// TwinCAT 3 PLC project ukazkaPlc
// Title: ukazkaPlc
// Company: TcOpen.MTS
// ProjectVersion: 0.6.0.913
// ProgramVersion: 3.1.4023.0
// libraries:
//   Tc2_Standard, * (Beckhoff Automation GmbH)
//   Tc2_System, * (Beckhoff Automation GmbH)
//   Tc3_Module, * (Beckhoff Automation GmbH)
//   TcoAbbRobotics, 0.11.0.71 (Vortex.Library)
//   TcoAbstractions, 0.11.0.71 (Vortex.Library)
//   TcoAimTtiPowerSupply, 0.11.0.71 (Vortex.Library)
//   TcoCognexVision, 0.11.0.71 (Vortex.Library)
//   TcoCore, 0.11.0.71 (Vortex.Library)
//   TcoData, 0.11.0.71 (Vortex.Library)
//   TcoDrivesBeckhoff, 0.11.0.71 (Vortex.Library)
//   TcoElements, 0.11.0.71 (Vortex.Library)
//   TcoInspectors, 0.11.0.71 (Vortex.Library)
//   TcoIo, 0.11.0.71 (Vortex.Library)
//   TcoKukaRobotics, 0.11.0.71 (Vortex.Library)
//   TcoMitsubishiRobotics, 0.11.0.71 (Vortex.Library)
//   TcoPneumatics, 0.11.0.71 (Vortex.Library)
//   TcoRexrothPress, 0.11.0.71 (Vortex.Library)
//   TcoTixonFeeding, 0.11.0.71 (Vortex.Library)
//   TcoUrRobotics, 0.11.0.71 (Vortex.Library)
//   TcoUtilities, 0.11.0.71 (Vortex.Library)
// project tree:
//   Abstractions/Components/ArrayRenderingExample/ SampleArrayToRender.TcDUT, SampleDataItem.TcDUT
//   Abstractions/Components/MtsFeeding/ TcoFeedingSequenceTask.TcPOU, TcoPlsPaletizator.TcPOU, TcoPlsPaletizator_Components.TcDUT, TcoPlsPaletizator_Config_v_1_x_x.TcDUT, TcoPlsPaletizator_Control_v_1_x_x.TcDUT, TcoPlsPaletizator_Status_v_1_x_x.TcDUT
//   Abstractions/Components/WrappedComponent/ WrappedComponentExample.TcPOU, WrappedComponentExample_Config.TcDUT, WrappedComponentExample_Control.TcDUT, WrappedComponentExample_Status.TcDUT, WrappedComponentsExample.TcDUT
//   Abstractions/CUBase/ CuBaseRecurringFail.TcDUT, CuBaseRecurringFailures.TcDUT, CUBase.TcPOU, CUBaseStatusInfo.TcDUT, CUBaseSettings.TcDUT, CUComponentsBase.TcDUT, ICUBase.TcIO, ICUTask.TcIO, OperatorInfo.TcDUT
//   Abstractions/CUBase/Data/ CuHeader.TcDUT, CUProcessDataBase.TcDUT, CUTechnologicalDataBase.TcDUT, eCUMode.TcDUT, eCUState.TcDUT, eDataEntityInvokeType.TcDUT, EntityHeader.TcDUT
//   Abstractions/CUBase/RemoteTasks/ ProductionPlaner.TcPOU
//   Abstractions/CUBase/Tasks/ CUBaseAutomat.TcPOU, CUBaseSuspend.TcPOU, CUBaseGround.TcPOU, CUBaseRecover.TcPOU
//   Abstractions/Generic/NotificationPanel/ NotificationPanel.TcPOU, NotificationPanelInfo.TcDUT
//   Abstractions/Safety/ControlButtons/ TcoControlButtons.TcPOU, ITcoControlButtons.TcIO, TcoControledZone_Info.TcDUT
//   Abstractions/Safety/ControlledZone/ TcoControlledZoneActionTask.TcPOU, TcoControlledZone.TcPOU, TcoControlledZone_Config.TcDUT, TcoControlledZone_Status.TcDUT
//   Abstractions/Safety/ControlVoltage/ ITcoControlVoltage.TcIO, TcoControlVoltage.TcPOU
//   Abstractions/Safety/DoorCircuit/ TcoDoorCircuit_Status.TcDUT, TcoDoorCircuit_Config.TcDUT, TcoDoorCircuit.TcPOU, ITcoDoorCircuit.TcIO
//   Abstractions/Safety/Doors/ ITcoDoorLock.TcIO, TcoStandardDoor.TcPOU, TcoBasicDoor.TcPOU
//   Abstractions/Safety/Estop/ TcoEmergencyStop.TcPOU
//   Abstractions/Safety/KeyMode/ TcoKeyMode_Config.TcDUT, TcoKeyMode_Status.TcDUT, TcoKeyMode.TcPOU, ITcoKeyMode.TcIO
//   Abstractions/Safety/KeyNormalService/ TcoKeyNormalService.TcPOU, ITcoKeyNormalSevice.TcIO
//   Abstractions/TcoCore/ CycleTimeAnalitics.TcDUT, TcoInnerTask.TcPOU, TcoTaskedSequencer.TcPOU, TcoTaskedService.TcPOU
//   Abstractions/Technology/ eStations.TcDUT
//   / MAIN.TcPOU, PlcTask.TcTTO
//   Technology/CU00x/Automat/ CU00xAutomatParalell_1_Task.TcPOU, CU00xAutomatTask.TcPOU
//   Technology/CU00x/Components/ CU00xExamplesOfComponents.TcDUT, CU00xComponents.TcDUT
//   Technology/CU00x/Data/ CU00xTechnologicalData.TcDUT, CU00xDialogContent.TcPOU, CU00xProcessData.TcDUT
//   Technology/CU00x/Ground/ CU00xGroundTask.TcPOU
//   Technology/CU00x/Manual/ CU00xManualTask.TcPOU
//   Technology/CU00x/Positions/ CU00xTestMultiPositions.TcPOU, Cu00xTestPositions.TcPOU
//   Technology/CU00x/Safety/Suspend/ CU00xSuspendTask.TcPOU
//   Technology/CU00x/Safety/Recover/ CU00xRecoverTask.TcPOU
//   Technology/Data/ ProcessData.TcDUT, ProcessDataManager.TcPOU, TcoEntityBase.TcDUT, TechnologicalDataManager.TcPOU, TechnologyData.TcDUT
//   Technology/CU00x/ CU00x.TcPOU
//   Technology/ Technology.TcPOU, TechnologyComponents.TcDUT (not stored)
//   DUTs/IO/PDOs/ Device_State_F0482DC3.TcDUT, Device_Control_6258066A.TcDUT, Inputs_23559BB0.TcDUT, Outputs_FC2FACAD.TcDUT, Modules_85784B27.TcDUT, Channel_830843C1.TcDUT, Channel_42CA91F7.TcDUT
//   DUTs/IO/Boxes/ EK1200_013D0B49.TcDUT, EK1122_1FC0878B.TcDUT, AES_510494FB.TcDUT, EPP1322_1FC0878B.TcDUT, EPP1809_32157CFD.TcDUT, EPP1008_78E8D3DD.TcDUT, EL1809_32157CFD.TcDUT, EL2809_2B6483BD.TcDUT, EL9011_D65D3D32.TcDUT
//   DUTs/IO/Devices/ SyncUnitTasks_4BE01469.TcDUT, SyncUnits_67D36DDA.TcDUT
//   DUTs/IO/Topology/ EK_E812B8FA.TcDUT, EC_4E5C738F.TcDUT, EC_245FBB9A.TcDUT
//   GVLs/ GVL_iXlinker.TcGVL
// real-time tasks:
//   TASK PlcTask: cycle T#10ms, priority 20, ADS port 350
//   TASK PlcTask1: cycle T#10ms, priority 21, ADS port 351
// I/O:
//   DEVICE EC1 (disabled), AmsNetId 172.20.21.220.7.1
//     (EK1200) [EK1200-5000 EtherCAT Power supply (2A E-Bus)]
//       EC (EK1122) [EK1122 2 port EtherCAT junction]
//       PN (EL6631) [EL6631 PROFINET IO Controller]
//       IA1 (EL1809) [EL1809 16Ch. Dig. Input 24V, 3ms]
//       QA1 (EL2809) [EL2809 16Ch. Dig. Output 24V, 0.5A]
//       Term 6 (EL4004) [EL4004 4Ch. Ana. Output 0-10V, 12bit]
//       Term 7 (EL7342) [EL7342 2Ch. DC motor output stage (50V, 3.5A)]
//       Term 8 (EL4004) [EL4004 4Ch. Ana. Output 0-10V, 12bit]
//       Term 9 (EL6001) [EL6001 Interface (RS232)]
//       Term 13 (EL9011) [EL9011 End Terminal]
//   DEVICE EC (disabled), AmsNetId 172.20.21.220.2.1
//     EC [EK1200-5000 EtherCAT Power supply (2A E-Bus)]
//       EK [EK1122 2 port EtherCAT junction]
//         PNEU [AES Fieldbus Coupler Gen2]
//           modules: Modules
//         AB [EPP1322-0001 3 port EtherCAT P gateway]
//         AB21 [EPP1809-0021 16 Ch. Dig. Input 24V, 3ms, M8]
//         AB22 [EPP1809-0021 16 Ch. Dig. Input 24V, 3ms, M8]
//         AB23 [EPP1008-0001 8 Ch. Dig. Input 24V, 3ms, M8]
//         AB24 [EPP1008-0001 8 Ch. Dig. Input 24V, 3ms, M8]
//       IA1 [EL1809 16Ch. Dig. Input 24V, 3ms]
//       QA1 [EL2809-0015 16Ch. Dig. Output 24V DC, 0.35A, not short-circuit proof]
//       Term 11 (EL9011) [EL9011 End Terminal]

CONFIGURATION ukazkaPlc
    RESOURCE PLC ON TwinCAT3
        TASK PlcTask(INTERVAL := T#10ms, PRIORITY := 20);
        PROGRAM MAIN WITH PlcTask : MAIN;
    END_RESOURCE
END_CONFIGURATION

// ---- Abstractions/Components/ArrayRenderingExample/SampleArrayToRender.TcDUT
TYPE SampleArrayToRender :
STRUCT
	Data	:	ARRAY  [0..100] OF SampleDataItem;
END_STRUCT
END_TYPE

// ---- Abstractions/Components/ArrayRenderingExample/SampleDataItem.TcDUT
TYPE SampleDataItem :
STRUCT
 	Measured : BOOL;
    Overrided : BOOL;
    Marginal : BOOL;
    FinalResults : BOOL;
END_STRUCT
END_TYPE

// ---- Abstractions/Components/MtsFeeding/TcoPlsPaletizator_Components.TcDUT
TYPE TcoPlsPaletizator_Components EXTENDS TcoCore.TcoStruct:
STRUCT
	
	{attribute wpf [Container(Layout.Stack)]}
	{attribute addProperty Name "(I1) <#Pritomnost blistra v presuvaci#>"}
	I1_PresentBlisterEntry : TcoElements.TcoDi(THISSTRUCT);
	
	{attribute addProperty Name "(I2) <#Pritomnost medzery medzi blistrami#>"}
	I2_PresentBlisterEntryEmptySpace : TcoElements.TcoDi(THISSTRUCT);
	
	{attribute addProperty Name "(I3) <#Zasobik blistrov prazdny#>"}
	I3_PresentBlistersInBufferEmpty : TcoElements.TcoDi(THISSTRUCT);

	
	{attribute addProperty Name "(I4) <#Pritomnost blistra v pracovnej pozicii#>"}
	I4_PresentBlisterInWorkingPos : TcoElements.TcoDi(THISSTRUCT);
		
	{attribute addProperty Name "(I5) <#Vystupny blister neje v sklzovom dopravniku#>"}
	I5_OutBlistersIsThrowedCorrectly : TcoElements.TcoDi(THISSTRUCT);
	
	{attribute addProperty Name "(I6) <#Vystupny blister snimanie vo vytahu#>"}
	I6_OutBlistersLisftSignal : TcoElements.TcoDi(THISSTRUCT);
	
	{attribute addProperty Name "(I7) <#Vystupny blister je nad Bufferom#>"}
	I7_OutBlistersIsAboveOutBuffer : TcoElements.TcoDi(THISSTRUCT);
	
	{attribute addProperty Name "(I8) <#Vystupny zasobnik je plny#>"}
	I8_OutBlistersBufferIsFull : TcoElements.TcoDi(THISSTRUCT);
	
	
	{attribute wpf [Container(Layout.Stack)]}
	{attribute addProperty Name "(P1) <#Vertikalny prisun vstupnych blistrov#>"}
	P1_VerticalSepareEntryBlisters : TcoPneumatics.TcoCylinder(THISSTRUCT);
	
	{attribute addProperty Name "(P2) <#Vertikalny prisun vstupnych blistrov#>"}
	P2_VerticalSepareEntryBlisters : TcoPneumatics.TcoCylinder(THISSTRUCT);
	
	{attribute addProperty Name "(P3) (P3.1) <#Horizontalny prisun vstupnych blistrov#>"}
	P3_HorizontalSepareEntryBlisters : TcoPneumatics.TcoDoubleCylinder(THISSTRUCT);
		
	{attribute addProperty Name "(P4) <#Prisun vstupneho blistra#>"}
	P4_FeedEntryBlister :TcoPneumatics.TcoCylinder(THISSTRUCT);
	
	{attribute addProperty Name "(P5) (P5.1)<#Horizontalny prisun vystupnych blistrov#>"}
	P5_HorizontalSepareOutBlisters : TcoPneumatics.TcoDoubleCylinder(THISSTRUCT);
	
	{attribute addProperty Name "(P6)<#Vertikalny prisun vystupnych blistrov#>"}
	P6_VerticalSepareOutBlister : TcoPneumatics.TcoCylinder(THISSTRUCT);
	
	{attribute addProperty Name "(P7) <#Podopretie vstupneho blistra#>"}
	P7_SupportEntryBlister : TcoPneumatics.TcoCylinder(THISSTRUCT);
	
	{attribute addProperty Name "(P8) (P8.1) <#Upevnenie zboku vstupneho blistra#>"}
	P8_FixEntryBlisterSide : TcoPneumatics.TcoDoubleCylinder(THISSTRUCT);
	
	{attribute addProperty Name "(P9) (P9.1) <#Zamknutue zhora vstupneho blistra#>"}
	P9_LockEntryBlisterTop : TcoPneumatics.TcoDoubleCylinder(THISSTRUCT);
	
	{attribute addProperty Name "(P10) (P10.1)<#Odelovac blistrov na vstupe#>"}
	P10_HoldEntrySepareOutBlister : TcoPneumatics.TcoDoubleCylinder(THISSTRUCT);
	
	
	
	{attribute wpf [Container(Layout.Stack,"Vseobecne")]}
	
	{attribute addProperty Name "(Q1) <#Signalizacia upozornenia R#>"}
	Q1_AttentionSignalisationR : TcoElements.TcoDo(THISSTRUCT);
	{attribute addProperty Name "(Q2) <#Signalizacia upozornenia G#>"}
	Q2_AttentionSignalisationG : TcoElements.TcoDo(THISSTRUCT);
	{attribute addProperty Name "(Q3) <#Signalizacia upozornenia B#>"}
	Q3_AttentionSignalisationB : TcoElements.TcoDo(THISSTRUCT);

	
	
END_STRUCT
END_TYPE

// ---- Abstractions/Components/MtsFeeding/TcoPlsPaletizator_Config_v_1_x_x.TcDUT
TYPE
    TcoPlsPaletizator_Config_v_1_x_x EXTENDS TcoCore.TcoStruct :
    STRUCT

	
        {attribute addProperty Name "<#Stabilizacny cas#>"}
		StabilisationTime : TIME :=T#500MS;
		{attribute addProperty Name "<#Blink period#>"}
		BlinkTime : TIME := T#500MS;
		
        {attribute addProperty Name "<#Zamykanie blistra zhora neaktive (P9)(P9.1)je nepritomne#>"}
		LockBlisterInPickPosInactive : BOOL;
		
		{attribute addProperty Name "<#Oddelovanie blistrov na vstupe neaktive (P10)(P10.1)je nepritomne#>"}
		SepareBlistersAtEntryInactive : BOOL;
    END_STRUCT
END_TYPE

// ---- Abstractions/Components/MtsFeeding/TcoPlsPaletizator_Control_v_1_x_x.TcDUT
TYPE TcoPlsPaletizator_Control_v_1_x_x EXTENDS TcoCore.TcoStruct:
STRUCT

		
END_STRUCT
END_TYPE

// ---- Abstractions/Components/MtsFeeding/TcoPlsPaletizator_Status_v_1_x_x.TcDUT
TYPE
    TcoPlsPaletizator_Status_v_1_x_x EXTENDS TcoCore.TcoStruct :
    STRUCT

        ActionDescription : STRING;
        SafeCondition : BOOL;
		EntryBufferEmpty:BOOL;
        BlisterReady : BOOL;
        OutBufferFull : BOOL;
    END_STRUCT
END_TYPE

// ---- Abstractions/Components/WrappedComponent/WrappedComponentExample_Config.TcDUT
TYPE
    WrappedComponentExample_Config EXTENDS TcoCore.TcoStruct :
    STRUCT

        VacuumReachedStabilisation : TIME := T#100MS;
        VacuumPushTime : TIME := T#100MS;
    END_STRUCT
END_TYPE

// ---- Abstractions/Components/WrappedComponent/WrappedComponentExample_Control.TcDUT
TYPE WrappedComponentExample_Control EXTENDS TcoCore.TcoStruct:
STRUCT

		Setpoint:INT;
		
END_STRUCT
END_TYPE

// ---- Abstractions/Components/WrappedComponent/WrappedComponentExample_Status.TcDUT
TYPE WrappedComponentExample_Status EXTENDS TcoCore.TcoStruct:
STRUCT

		ProgressThrow:INT;
		ActionDescription:STRING;
END_STRUCT
END_TYPE

// ---- Abstractions/Components/WrappedComponent/WrappedComponentsExample.TcDUT
TYPE WrappedComponentsExample EXTENDS TcoCore.TcoStruct:
STRUCT
	
		{attribute addProperty Name "Vacuum Reached"}
		VacuumReached : TcoElements.TcoDi(THISSTRUCT);
		{attribute addProperty Name "Vacuum On"}
		VacuumOn : TcoElements.TcoDo(THISSTRUCT);
		{attribute addProperty Name "Vacuum Push"}
		VacuumPush : TcoElements.TcoDo(THISSTRUCT);
		
		{attribute addProperty Name "Gripper"}
		Gripper : TcoPneumatics.TcoCylinder(THISSTRUCT);
  
		{attribute addProperty Name "Manipulator"}
		Manipulator : TcoDrivesBeckhoff.TcoMultiAxis(THISSTRUCT);

		{attribute addProperty Name "Component Picked"}
		PresenceInGripper : TcoElements.TcoDi(THISSTRUCT);

	
	
END_STRUCT
END_TYPE

// ---- Abstractions/CUBase/CuBaseRecurringFail.TcDUT
TYPE CuBaseRecurringFail :
STRUCT
	Reached:BOOL;
	Result:TcoComprehensiveResult;
	Counter:UINT;
	
	
	
	
	
END_STRUCT
END_TYPE

// ---- Abstractions/CUBase/CuBaseRecurringFailures.TcDUT
TYPE CuBaseRecurringFailures EXTENDS TcoCore.TcoStruct : 
	STRUCT
   		AnyRecurringFails : CuBaseRecurringFail;
    	SameRecurringFails : CuBaseRecurringFail;
	END_STRUCT
END_TYPE

// ---- Abstractions/CUBase/CUBaseStatusInfo.TcDUT
TYPE
    CUBaseStatusInfo EXTENDS TcoCore.TcoStruct :
    STRUCT
     Mode                   : eCUMode;
     CurrentTaskDescription : STRING;
     CurrentUid             : INT;
     CurrentOperation       : STRING(255);
     CurrentCycleTime       : TIME;
	 AverageCycleTime       : TIME;
     CurrentIsInStepMode    : BOOL;
     CurrentCleanCycleTime  : TIME;
	 AverageCleanCycleTime  : TIME;
     State	                : eCUState;
     InSavingEnergy         : BOOL;
    END_STRUCT
END_TYPE

// ---- Abstractions/CUBase/CUBaseSettings.TcDUT
TYPE CUBaseSettings EXTENDS TcoCore.TcoStruct : STRUCT
    DeafultCycleTime : TIME;
    WarningCycleTime : TIME;
    ErrorCycleTime : TIME;
    SaveEnergyTime : TIME;
    AnyRecurringFailure : UINT;
    SameRecurringFailure : UINT;
END_STRUCT
END_TYPE

// ---- Abstractions/CUBase/CUComponentsBase.TcDUT
TYPE
    CUComponentsBase EXTENDS TcoCore.TcoStruct :
    STRUCT
       
    END_STRUCT
END_TYPE

// ---- Abstractions/CUBase/Data/CuHeader.TcDUT
TYPE CuHeader EXTENDS TcoCore.TcoStruct :
STRUCT
	{attribute addProperty Name "<#Next on Passed#>"}
	NextOnPassed : eStations;
	{attribute addProperty Name "<#Next on Failed#>"}
	NextOnFailed : eStations;
	{attribute clr [RenderIgnore("Control", "ShadowControl")]}
	{attribute addProperty Name "<#Cycle time#>"}
	CycleTime : TIME;
	{attribute clr [RenderIgnore("Control", "ShadowControl")]}
	{attribute addProperty Name "<#Clean loop time#>"}
	CleanLoopTime : TIME;
	{attribute clr [RenderIgnore("Control", "ShadowControl")]}
	{attribute addProperty Name "<#Operation started#>"}
	OperationsStarted : DT;
	{attribute clr [RenderIgnore("Control", "ShadowControl")]}
	{attribute addProperty Name "<#Operation ended#>"}
	OperationsEnded : DT;	
	{attribute clr [RenderIgnore("Control", "ShadowControl")]}
	{attribute addProperty Name "<#Operator#>"}
	Operator :STRING;	
END_STRUCT
END_TYPE

// ---- Abstractions/CUBase/Data/CUProcessDataBase.TcDUT
{attribute clr [Container(Layout.Stack)]}
{attribute clr [Group(Layout.Scroll)]}
TYPE CUProcessDataBase EXTENDS TcoCore.TcoStruct :
STRUCT
	{attribute wpf [Container(Layout.Stack)]}
	{attribute wpf [Group(Layout.GroupBox)]}
	Header : CuHeader := (Parent := THISSTRUCT);
END_STRUCT
END_TYPE

// ---- Abstractions/CUBase/Data/CUTechnologicalDataBase.TcDUT
{attribute clr [Container(Layout.Stack)]}
{attribute clr [Group(Layout.Scroll)]}
TYPE CUTechnologicalDataBase EXTENDS TcoCore.TcoStruct :
STRUCT
	{attribute wpf [Container(Layout.Stack,"General")]}
	{attribute wpf [Group(Layout.GroupBox)]}
	{attribute addProperty Name "<#Cycle time#> - <#Nominal#>"}
	IdealCycleTime   : TIME;
	
	
	{attribute addProperty Name "<#Cycle time#> - <#Warning#>"}
	WarningCycleTime : TIME;
    
	{attribute addProperty Name "<#Cycle time#> - <#Error#>"}
	ErrorCycleTime   : TIME;

	
	{attribute addProperty Name "<#Step time#> - <#Warning#>"}
	WarningStepAlarmTime : TIME;
    
	{attribute addProperty Name "<#Step time#> - <#Error#>"}
	ErrorStepAlarmTime   : TIME;
	
	{attribute addProperty Name "<#Energy saving mode - Inactivity time#>"}
	TimeToEntryEnergySavingMode : TIME;
	
	
	
	(*~
	<docu>
		<summary>
			The maximum allowed number of the any (arbitrary) recuring (consecutive)  failures.
		</summary>			
	</docu>	
	~*)
	{attribute addProperty Name "<#Max allowed number of any recurring failures (consecutive)#>"}
	AnyRecurringFailure   : UINT;
	
	

	(*~
	<docu>
		<summary>
			The maximum allowed number of the same (identical) recuring (consecutive) failures. 
		</summary>			
	</docu>	
	~*)
	{attribute addProperty Name "<#Max allowed number of same recurring failures (consecutive)#>"}
	SameRecurringFailure   : UINT;
	
	
END_STRUCT
END_TYPE

// ---- Abstractions/CUBase/Data/eCUMode.TcDUT
{attribute 'qualified_only'}
{attribute 'strict'}
TYPE
    eCUMode :
    (
        NoMode         := 0,
        GroundMode     := 10,
        GroundModeDone := 15,
        AutomatMode    := 20,
        ManualMode     := 30
    );
END_TYPE

// ---- Abstractions/CUBase/Data/eCUState.TcDUT
{attribute 'qualified_only'}
{attribute 'strict'}
TYPE
    eCUState :
    (
        None       := 0,
        HasWarning := 10,
        HasError   := 20
    );
END_TYPE

// ---- Abstractions/CUBase/Data/eDataEntityInvokeType.TcDUT
{attribute 'qualified_only'}
{attribute 'strict'}
TYPE eDataEntityInvokeType : (
    InvokeAndWaitDone := 0,
    InvokeOnly	 := 10
);
END_TYPE

// ---- Abstractions/CUBase/Data/EntityHeader.TcDUT
{attribute wpf [Container(Layout.Stack)]}
{attribute wpf [Group(Layout.Scroll)]}
{attribute addProperty Name "<#Entity header#>"}
TYPE
    EntityHeader EXTENDS TcoCore.TcoStruct :
    STRUCT
        {attribute addProperty Name "<#Recipe#>"}
        {attribute clr [RenderIgnore("Control", "ShadowControl")]}
        Recipe : STRING(255);
        {attribute addProperty Name "<#Recipe created#>"}
        {attribute clr [RenderIgnore("Control", "ShadowControl")]}
        RecipeCreated : DT;
        {attribute addProperty Name "<#Recipe modified#>"}
        {attribute clr [RenderIgnore("Control", "ShadowControl")]}
        RecipeLastModified : DT;
        {attribute addProperty Name "<#Carrier#>"}
        {attribute clr [RenderIgnore("Control", "ShadowControl")]}
        Carrier : STRING;
        {attribute addProperty Name "<#Reset#>"}
        {attribute clr [RenderIgnore("Control", "ShadowControl")]}
        WasReset : BOOL;
        {attribute addProperty Name "<#Master#>"}
        {attribute clr [RenderIgnore("Control", "ShadowControl")]}
        IsMaster : BOOL;
        {attribute addProperty Name "<#Empty#>"}
        {attribute clr [RenderIgnore("Control", "ShadowControl")]}
        IsEmpty : BOOL;
        {attribute addProperty Name "<#Last station#>"}
        LastStation : eStations;
        {attribute addProperty Name "<#Next station#>"}
        NextStation : eStations;
        {attribute addProperty Name "<#Operations opened#>"}
        OpenOn : eStations;
        {attribute addProperty Name "<#Results#>"}
        Results : TcoInspectors.TcoComprehensiveResult;

        {attribute addProperty Name "<#Reworked#>"}
        {attribute clr [RenderIgnore("Control", "ShadowControl")]}
         WasReworked : BOOL;

        {attribute addProperty Name "<#Last Rework Name#>"}
        {attribute clr [RenderIgnore("Control", "ShadowControl")]}
         LastReworkName : STRING;

        {attribute addProperty Name "<#Rework Count#>"}
        {attribute clr [RenderIgnore("Control", "ShadowControl")]}
        ReworkCount : SINT;

    END_STRUCT
END_TYPE

// ---- Abstractions/CUBase/OperatorInfo.TcDUT
TYPE OperatorInfo EXTENDS TcoCore.TcoStruct :
STRUCT
	UserName : STRING(255);
END_STRUCT
END_TYPE

// ---- Abstractions/Generic/NotificationPanel/NotificationPanelInfo.TcDUT
TYPE NotificationPanelInfo :
STRUCT
	{attribute addProperty Name "<#Control voltage#>"}
	ControlVoltage : BOOL;
	{attribute addProperty Name "<#Air pressure#>"}
	AirPressure : BOOL;
	{attribute addProperty Name "<#Autmatic mode allowed#>"}
	AutomatAllowed : BOOL;
	{attribute addProperty Name "<#Emergency stop#>"}
  	EmergencyStop : BOOL; 
	{attribute addProperty Name "<#Safety doors OK#>"}
  	SafetyDoorOk : BOOL;    
	{attribute addProperty Name "<#Doors closed#>"}
  	DoorClosed : BOOL;  
	{attribute addProperty Name "<#Doors locked#>"}
	DoorLocked : BOOL;
	{attribute addProperty Name "<#Light curtain#>"}
  	LightCurtain : BOOL;
	{attribute addProperty Name "<#Process data#>"}
  	ProcessDataOk : BOOL;
	{attribute addProperty Name "<#Technology data#>"}
  	TechnologyDataOk : BOOL;
END_STRUCT
END_TYPE

// ---- Abstractions/Safety/ControlButtons/TcoControledZone_Info.TcDUT
TYPE TcoControledZone_Info :
STRUCT
	{attribute addProperty Name "<#All#> - <#In automatic#>"}
	AllInAuto            : BOOL;
	
	{attribute addProperty Name "<#All#> - <#Is grounding#>"}
	AllInGrounding       : BOOL;
	
	{attribute addProperty Name "<#All#> - <#In manual#>"}
	AllInManual          : BOOL;
	
	{attribute addProperty Name "<#All#> - <#Idle#>"}
	AllIdle          : BOOL;

	{attribute addProperty Name "<#All#> - <#Grounded#>"}
	AllGrounded          : BOOL;
	
	{attribute addProperty Name "<#All#> - <#In step mode#>"}
	AllInStepMode        : BOOL;
	
	{attribute addProperty Name "<#All#> - <#Recovered#>"}
	AllRecovered        : BOOL;
	
	{attribute addProperty Name "<#All#> - <#Suspended#>"}
	AllSuspended        : BOOL;
	
	{attribute addProperty Name "<#All#> - <#Holding process#>"}
	AllHolding           : BOOL;
	
	{attribute addProperty Name "<#All#> - <#In Inactive or Manual or Grounded#>"}
	AllInactiveOrManualOrGrounded  : BOOL;
	
	{attribute addProperty Name "<#Group#> - <#Any station in automatic mode#>"}
	AnyInAuto            : BOOL;
	
	{attribute addProperty Name "<#Group#> - <#Any station in manual mode#>"}
	AnyInManual          : BOOL;
	
	{attribute addProperty Name "<#Group#> - <#Any station in step mode#>"}
	AnyInStepMode        : BOOL;
	
	{attribute addProperty Name "<#Group#> - <#Any station is grounding#>"}
	AnyGrounding         : BOOL;
	
	{attribute addProperty Name "<#Group#> - <#Any station is holded#>"}
	AnyInHolding         : BOOL;
	
	{attribute addProperty Name "<#Control panel#> - <#All keys in automatic#>"}
	AllKeysAuto          : BOOL;
	
	{attribute addProperty Name "<#Control panel#> - <#All keys in normal#>"}
	AllKeysNormal        : BOOL;
	
	{attribute addProperty Name "<#Control panel#> - <#Any key in manual#>"}
	AnyKeyManual         : BOOL;
	
	{attribute addProperty Name "<#Control panel#> - <#Any key in step#>"}
	AnyKeyStep           : BOOL;
	
	{attribute addProperty Name "<#Control panel#> - <#Any key in service#>"}
	AnyKeyService        : BOOL;
	
	{attribute addProperty Name "<#Control panel#> - <#Any button#> - <#Recover#>"}
	AnyButtonRecover       : BOOL;
	
	{attribute addProperty Name "<#Control panel#> - <#Any button#> - <#Suspend#>"}
	AnyButtonSuspend        : BOOL;
	
	{attribute addProperty Name "<#Control panel#> - <#Any button#> - <#Ground#>"}
	AnyButtonGround      : BOOL;
	
	{attribute addProperty Name "<#Control panel#> - <#Any button#> - <#Auto#>"}
	AnyButtonAuto     : BOOL;
	
	{attribute addProperty Name "<#Deadman#> - <#Any present#>"}
	AnyDeadmanPresent    : BOOL;

END_STRUCT
END_TYPE

// ---- Abstractions/Safety/ControlledZone/TcoControlledZone_Config.TcDUT
TYPE
    TcoControlledZone_Config :
    STRUCT
        MaxControledUnits : USINT := 12;
        MaxControlButtons : USINT := 4;
        MaxKeyMode : USINT := 4;
        MaxKeyNormalService : USINT := 4;
        DoorsLocked : TIME := T#1S;
		AirPressureErrorTime : TIME :=T#5S;
    END_STRUCT
END_TYPE

// ---- Abstractions/Safety/ControlledZone/TcoControlledZone_Status.TcDUT
TYPE TcoControlledZone_Status :
STRUCT
	ActionDescription : STRING(100);	
	State : TcoControledZone_Info;	
	
END_STRUCT
END_TYPE

// ---- Abstractions/Safety/DoorCircuit/TcoDoorCircuit_Status.TcDUT
TYPE TcoDoorCircuit_Status :
STRUCT
	ActionDescription : STRING(100);	
END_STRUCT
END_TYPE

// ---- Abstractions/Safety/DoorCircuit/TcoDoorCircuit_Config.TcDUT
TYPE
    TcoDoorCircuit_Config :
    STRUCT
        InfoTime : TIME := T#2S;
        ErrorTime : TIME := T#0S;
		MaxDoors : USINT:=12;
		MaxLocalDoorsVoltage : USINT:=4;
		MaxLocalVoltage: USINT:=4;
		MaxGlobalVoltage: USINT:=4;
	
    END_STRUCT
END_TYPE

// ---- Abstractions/Safety/KeyMode/TcoKeyMode_Config.TcDUT
TYPE
    TcoKeyMode_Config :
    STRUCT
        SwitKeyStanilisiation : TIME := T#500mS;

	
    END_STRUCT
END_TYPE

// ---- Abstractions/Safety/KeyMode/TcoKeyMode_Status.TcDUT
TYPE TcoKeyMode_Status :
STRUCT
	ActionDescription : STRING(100);	

END_STRUCT
END_TYPE

// ---- Abstractions/TcoCore/CycleTimeAnalitics.TcDUT
TYPE CycleTimeAnalitics :
STRUCT

	{attribute addProperty Name "<#Average cycle time#>"}
	Average:TIME;
	
	{attribute addProperty Name "<#Average clean cycle time#>"}
	AverageCleanCycle:TIME;
	
	{attribute addProperty Name "<#Average cycle time filter constant#>"}
	FilterConstant:UINT:=10;	
	

	
END_STRUCT
END_TYPE

// ---- Abstractions/Technology/eStations.TcDUT
{attribute 'qualified_only'}
{attribute 'strict'}
TYPE
    eStations :
    (
		CU00x := 100,
        ST_1  := 1,
        ST_2  := 2,
        ST_3  := 3,
        ST_4  := 4,
        ST_5  := 5,
        ST_6  := 6,
        ST_7  := 7,
        ST_8  := 8,
        ST_9  := 9,
        ST_10 := 10,
        ST_11 := 11,
        ST_12 := 12,
        ST_13 := 13,
        ST_14 := 14,
        ST_15 := 15,
        ST_16 := 16,
        ST_17 := 17,
        ST_18 := 18,
        ST_19 := 19,
        ST_20 := 20,
        NONE  := 32767
    );
END_TYPE

// ---- Technology/CU00x/Components/CU00xExamplesOfComponents.TcDUT
{attribute wpf [Container(Layout.Stack)]}	
{attribute wpf [Group(Layout.Scroll)]}
TYPE CU00xExamplesOfComponents EXTENDS TcoCore.TcoStruct:
STRUCT
		{attribute wpf [Container(Layout.Stack,"PNEU")]}	
		{attribute addProperty Name "(A1)HORIZONTAL AXIS"}
      	horizontalCylinder : TcoPneumatics.TcoCylinder(THISSTRUCT); 
		{attribute addProperty Name "(A2)VERTICAL AXIS"}
      	verticalCylinder : TcoPneumatics.TcoCylinder(THISSTRUCT); 
		
		{attribute addProperty Name "(A3)DOUBLE "}
      	doubleCylinder : TcoPneumatics.TcoDoubleCylinder(THISSTRUCT); 
		
		{attribute wpf [Container(Layout.Stack,"INPUTS")]}	
		{attribute addProperty Name "PRESENCE ON INSPECTION"}
     	PresenceOnInspection : TcoElements.TcoDi(THISSTRUCT);
		
		{attribute addProperty Name "PRESENCE AT ENTRY CONVEYOR"}
     	PresenceComponentAtEntr: TcoElements.TcoDi(THISSTRUCT);
		
		{attribute addProperty Name "COLISION SENSOR"}
     	ColisonSensorComponent: TcoElements.TcoDi(THISSTRUCT);

		{attribute addProperty Name "CONVEYOR AT ENTRY IS EMPTY"}
     	ConvAtEntryIsEmpty : TcoElements.TcoDi(THISSTRUCT);
		
		{attribute addProperty Name "INSPECTION NOK"}
     	InspectionIsNok : TcoElements.TcoDi(THISSTRUCT);
		

		{attribute wpf [Container(Layout.Stack,"OUTPUTS")]}		
		{attribute addProperty Name "LIGHT ON"}
     	LightOn : TcoElements.TcoDi(THISSTRUCT); 
		
		{attribute addProperty Name "LIGHT OFF"}
     	LightOff : TcoElements.TcoDi(THISSTRUCT);
		{attribute wpf [Container(Layout.Stack,"ANALOGS")]}	
		{attribute addProperty Name "VERIFY SETPOINT"}
     	VerifySetpoint : TcoElements.TcoAi(THISSTRUCT);
		{attribute addProperty Name "SETPOINT"}
     	Setpoint : TcoElements.TcoAo(THISSTRUCT);   
		
		{attribute addProperty Name "SampleDataToRender"}
     	ArrayToRender : SampleArrayToRender;   

END_STRUCT
END_TYPE

// ---- Technology/CU00x/Data/CU00xTechnologicalData.TcDUT
TYPE
    CU00xTechnologicalData EXTENDS CUTechnologicalDataBase : 
    STRUCT		
		{attribute wpf [Container(Layout.Stack,"Station specific data")]}
		{attribute wpf [Group(Layout.GroupBox)]}
		{attribute addProperty Name "Axis Home position"}
        ServoHomePosition : LREAL;
		{attribute addProperty Name "Axis Work position"}
		ServoWorkPosition : LREAL;
    END_STRUCT
END_TYPE

// ---- Technology/Data/ProcessData.TcDUT
{attribute clr [Container(Layout.Tabs)]}
TYPE
    ProcessData EXTENDS TcoEntityBase :
    STRUCT

        {attribute addProperty Name "<#Entity header#>"}
        EntityHeader : EntityHeader     := (Parent := THISSTRUCT);
		{attribute addProperty Name "<#CU00x#>"}
		{attribute clr [Container(Layout.Stack)]}
        CU00x : CU00xProcessData := (Parent := THISSTRUCT);
    END_STRUCT
END_TYPE

// ---- Technology/CU00x/Components/CU00xComponents.TcDUT
{attribute wpf [Container(Layout.Tabs)]}
TYPE
    CU00xComponents EXTENDS CUComponentsBase :
    STRUCT

		{attribute wpf [Container(Layout.Stack,"VSTUPY")]}	
		{attribute wpf [Group(Layout.Scroll)]}
		{attribute addProperty Name "Vstup 1"}   
		IN1 : TcoElements.TcoDi(THISSTRUCT);
		{attribute addProperty Name "Vstup 2"}  
		IN2 : TcoElements.TcoDi(THISSTRUCT);
		{attribute addProperty Name "Vstup 3"}  
		IN3 : TcoElements.TcoDi(THISSTRUCT);
		
		{attribute wpf [Container(Layout.Stack,"VÝSTUPY")]}	
		{attribute wpf [Group(Layout.Scroll)]}
		{attribute addProperty Name "Výstup 1"}   
		OUT1 : TcoElements.TcoDo(THISSTRUCT);
		{attribute addProperty Name "Výstup 2"}   
		OUT2 : TcoElements.TcoDo(THISSTRUCT);
		{attribute addProperty Name "Výstup 3"}   
		OUT3 : TcoElements.TcoDo(THISSTRUCT);


		{attribute wpf [Container(Layout.Stack,"PNEUMATIKA")]}	
		{attribute wpf [Group(Layout.Scroll)]}
		
		{attribute addProperty Name "Vertikálny piest"}                  
		{attribute addProperty _moveHomeDefaultName "<#MOVE DOWN#>"}    
		{attribute addProperty _moveWorkDefaultName "<#MOVE UP#>"} 
		{attribute addProperty _stopDefaultName "<#STOP#>"}             
		VerticalPiston : TcoPneumatics.TcoCylinder(THISSTRUCT);
		
		
		{attribute addProperty Name "Horizontálny piest"}                  
		{attribute addProperty _moveHomeDefaultName "<#MOVE DOWN#>"}    
		{attribute addProperty _moveWorkDefaultName "<#MOVE UP#>"} 
		{attribute addProperty _stopDefaultName "<#STOP#>"}             
		HorizontalPiston : TcoPneumatics.TcoCylinder(THISSTRUCT);
		
		{attribute addProperty Name "Dvojitý piest"}                  
		{attribute addProperty _moveHomeDefaultName "<#MOVE DOWN#>"}    
		{attribute addProperty _moveWorkDefaultName "<#MOVE UP#>"} 
		{attribute addProperty _stopDefaultName "<#STOP#>"}             
		DoublePiston : TcoPneumatics.TcoDoubleCylinder(THISSTRUCT);
		
	

		{attribute wpf [Container(Layout.Stack,"VISION")]}	
		{attribute wpf [Group(Layout.Scroll)]}
		{attribute addProperty Name "Dataman"}
     	Dmc : TcoCognexVision.TcoDataman_v_5_x_x(THISSTRUCT);

		{attribute wpf [Container(Layout.Stack,"ROBOTIKA")]}	
		{attribute wpf [Group(Layout.Scroll)]}
		{attribute addProperty Name "Abb IRC 5"}
     	AbbIrc5 : TcoAbbRobotics.TcoIrc5_v_1_x_x(THISSTRUCT);

		

    END_STRUCT
END_TYPE

// ---- Technology/CU00x/Data/CU00xProcessData.TcDUT
TYPE
    CU00xProcessData EXTENDS CUProcessDataBase :
    STRUCT
		{attribute wpf [Container(Layout.Stack)]}
        BoltPresenceInspector : TcoInspectors.TcoDigitalInspector(THISSTRUCT);
		BoltDimensionPresenceInspector : TcoInspectors.TcoAnalogueInspector(THISSTRUCT);
		BoltDatacodePresenceInspector : TcoInspectors.TcoDataInspector(THISSTRUCT);

		{attribute addProperty Name "Dimension inspection 1"}
        Dim_Inspector_1 : TcoInspectors.TcoAnalogueInspector(THISSTRUCT);
		{attribute addProperty Name "Dimension inspection 2"}
        Dim_Inspector_2 : TcoInspectors.TcoAnalogueInspector(THISSTRUCT);
		{attribute addProperty Name "Dimension inspection 3"}
		Dim_Inspector_3 : TcoInspectors.TcoAnalogueInspector(THISSTRUCT);
		{attribute addProperty Name "Dimension inspection 4"}
        Dim_Inspector_4 : TcoInspectors.TcoAnalogueInspector(THISSTRUCT);
		{attribute addProperty Name "Dimension inspection 5"}
        Dim_Inspector_5 : TcoInspectors.TcoAnalogueInspector(THISSTRUCT);
		{attribute addProperty Name "Dimension inspection 6"}
        Dim_Inspector_6 : TcoInspectors.TcoAnalogueInspector(THISSTRUCT);
		{attribute addProperty Name "Dimension inspection 7"}
        Dim_Inspector_7 : TcoInspectors.TcoAnalogueInspector(THISSTRUCT);
		{attribute addProperty Name "Dimension inspection 8"}
        Dim_Inspector_8 : TcoInspectors.TcoAnalogueInspector(THISSTRUCT);
		{attribute addProperty Name "Dimension inspection 9"}
        Dim_Inspector_9 : TcoInspectors.TcoAnalogueInspector(THISSTRUCT);
		{attribute addProperty Name "Dimension inspection 10"}
        Dim_Inspector_10 : TcoInspectors.TcoAnalogueInspector(THISSTRUCT);
		
		{attribute addProperty Name "Dimension inspection 11"}
        Dim_Inspector_11 : TcoInspectors.TcoAnalogueInspector(THISSTRUCT);
		{attribute addProperty Name "Dimension inspection 12"}
        Dim_Inspector_12 : TcoInspectors.TcoAnalogueInspector(THISSTRUCT);
		{attribute addProperty Name "Dimension inspection 13"}
		Dim_Inspector_13 : TcoInspectors.TcoAnalogueInspector(THISSTRUCT);
		{attribute addProperty Name "Dimension inspection 14"}
        Dim_Inspector_14 : TcoInspectors.TcoAnalogueInspector(THISSTRUCT);
		{attribute addProperty Name "Dimension inspection 15"}
        Dim_Inspector_15 : TcoInspectors.TcoAnalogueInspector(THISSTRUCT);
		{attribute addProperty Name "Dimension inspection 16"}
        Dim_Inspector_16 : TcoInspectors.TcoAnalogueInspector(THISSTRUCT);
		{attribute addProperty Name "Dimension inspection 17"}
        Dim_Inspector_17 : TcoInspectors.TcoAnalogueInspector(THISSTRUCT);
		{attribute addProperty Name "Dimension inspection 18"}
        Dim_Inspector_18 : TcoInspectors.TcoAnalogueInspector(THISSTRUCT);
		{attribute addProperty Name "Dimension inspection 19"}
        Dim_Inspector_19 : TcoInspectors.TcoAnalogueInspector(THISSTRUCT);
		{attribute addProperty Name "Dimension inspection 20"}
        Dim_Inspector_20 : TcoInspectors.TcoAnalogueInspector(THISSTRUCT);
    END_STRUCT
END_TYPE

// ---- Technology/Data/TcoEntityBase.TcDUT
TYPE TcoEntityBase EXTENDS TcoData.TcoEntity :
STRUCT
	{attribute clr [RenderIgnore("Control", "ShadowControl")]}
	{attribute addProperty Name "<#Created#>"}
	_Created : DT;
	{attribute clr [RenderIgnore("Control", "ShadowControl")]}
	{attribute addProperty Name "<#Modified#>"}
	_Modified : DT;
END_STRUCT
END_TYPE

// ---- Technology/Data/TechnologyData.TcDUT
{attribute clr [Container(Layout.Tabs)]}
TYPE
    TechnologyData EXTENDS TcoEntityBase :
    STRUCT

        CU00x : CU00xTechnologicalData := (Parent := THISSTRUCT);
    END_STRUCT
END_TYPE

// ---- DUTs/IO/PDOs/Device_State_F0482DC3.TcDUT
{attribute 'GeneratedUsingTerminal: AES-D-BC-ECAT Gen2-0001'}
{attribute addProperty BoxType "AES-D-BC-ECAT Gen2-0001"}
{attribute addProperty Id "IO_1_8AT %I*BYTE1IO_9_10AT %I*BYTE1ValveExtSupplyDiag_1_6AT %I*BYTE1Undervoltage_UAAT %I*BOOL1UA_OFFAT %I*BOOL1Undervoltage_ULAT %I*BOOL1UL_OFFAT %I*BOOL1Undervoltage_5VAT %I*BOOL1CommonValveAT %I*BOOL1Configuration_Error_ValveAT %I*BOOL1Configuration_Error_IO_ModuleAT %I*BOOL1Switchcounter_ErrorAT %I*BOOL1Configuratipn_Error_SLSAT %I*BOOL1Heardbeat_xAT %I*BOOL1Unknown_Module_IDAT %I*BOOL1Count_IO_Module_to_bigAT %I*BOOL1"}
{attribute addProperty CRC "4031262147"}
{attribute addProperty Size "16"}
TYPE Device_State_F0482DC3 EXTENDS TcoIo.InputBase_8311D824 :
STRUCT
	{attribute addProperty Name "IO_1_8"}
	IO_1_8 AT %I* : BYTE;
	{attribute addProperty Name "IO_9_10"}
	IO_9_10 AT %I* : BYTE;
	{attribute addProperty Name "ValveExtSupplyDiag_1_6"}
	ValveExtSupplyDiag_1_6 AT %I* : BYTE;
	{attribute addProperty Name "Undervoltage_UA"}
	Undervoltage_UA AT %I* : BOOL;
	{attribute addProperty Name "UA_OFF"}
	UA_OFF AT %I* : BOOL;
	{attribute addProperty Name "Undervoltage_UL"}
	Undervoltage_UL AT %I* : BOOL;
	{attribute addProperty Name "UL_OFF"}
	UL_OFF AT %I* : BOOL;
	{attribute addProperty Name "Undervoltage_5V"}
	Undervoltage_5V AT %I* : BOOL;
	{attribute addProperty Name "CommonValve"}
	CommonValve AT %I* : BOOL;
	{attribute addProperty Name "Configuration_Error_Valve"}
	Configuration_Error_Valve AT %I* : BOOL;
	{attribute addProperty Name "Configuration_Error_IO_Module"}
	Configuration_Error_IO_Module AT %I* : BOOL;
	{attribute addProperty Name "Switchcounter_Error"}
	Switchcounter_Error AT %I* : BOOL;
	{attribute addProperty Name "Configuratipn_Error_SLS"}
	Configuratipn_Error_SLS AT %I* : BOOL;
	{attribute addProperty Name "Heardbeat_x"}
	Heardbeat_x AT %I* : BOOL;
	{attribute addProperty Name "Unknown_Module_ID"}
	Unknown_Module_ID AT %I* : BOOL;
	{attribute addProperty Name "Count_IO_Module_to_big"}
	Count_IO_Module_to_big AT %I* : BOOL;
END_STRUCT
END_TYPE

// ---- DUTs/IO/PDOs/Device_Control_6258066A.TcDUT
{attribute 'GeneratedUsingTerminal: AES-D-BC-ECAT Gen2-0001'}
{attribute addProperty BoxType "AES-D-BC-ECAT Gen2-0001"}
{attribute addProperty Id "Web_App_DisableAT %Q*BOOL1Freeze_OutputAT %Q*BOOL1HL_SwapAT %Q*BOOL1Default_Modul_ControlAT %Q*BOOL1"}
{attribute addProperty CRC "1649935978"}
{attribute addProperty Size "4"}
TYPE Device_Control_6258066A EXTENDS TcoIo.OutputBase_10CEE7DE :
STRUCT
	{attribute addProperty Name "Web_App_Disable"}
	Web_App_Disable AT %Q* : BOOL;
	{attribute addProperty Name "Freeze_Output"}
	Freeze_Output AT %Q* : BOOL;
	{attribute addProperty Name "HL_Swap"}
	HL_Swap AT %Q* : BOOL;
	{attribute addProperty Name "Default_Modul_Control"}
	Default_Modul_Control AT %Q* : BOOL;
END_STRUCT
END_TYPE

// ---- DUTs/IO/PDOs/Inputs_23559BB0.TcDUT
{attribute 'GeneratedUsingTerminal: AES-D-BC-ECAT Gen2-0001'}
{attribute addProperty BoxType "AES-D-BC-ECAT Gen2-0001"}
{attribute addProperty Id "digital_Data_IAT %I*ARRAY[0..31] OF USINT32"}
{attribute addProperty CRC "1374483313"}
{attribute addProperty Size "32"}
TYPE Inputs_23559BB0 EXTENDS TcoIo.InputBase_8311D824 :
STRUCT
	{attribute addProperty Name "digital_Data_I"}
	digital_Data_I AT %I* : ARRAY[0..31] OF USINT;
END_STRUCT
END_TYPE

// ---- DUTs/IO/PDOs/Outputs_FC2FACAD.TcDUT
{attribute 'GeneratedUsingTerminal: AES-D-BC-ECAT Gen2-0001'}
{attribute addProperty BoxType "AES-D-BC-ECAT Gen2-0001"}
{attribute addProperty Id "digital_Data_OAT %Q*ARRAY[0..31] OF USINT32"}
{attribute addProperty CRC "2024821696"}
{attribute addProperty Size "32"}
TYPE Outputs_FC2FACAD EXTENDS TcoIo.OutputBase_10CEE7DE :
STRUCT
	{attribute addProperty Name "digital_Data_O"}
	digital_Data_O AT %Q* : ARRAY[0..31] OF USINT;
END_STRUCT
END_TYPE

// ---- DUTs/IO/PDOs/Modules_85784B27.TcDUT
{attribute 'GeneratedUsingTerminal: AES-D-BC-ECAT Gen2-0001'}
{attribute addProperty BoxType "AES-D-BC-ECAT Gen2-0001"}
{attribute addProperty Id "InputsInputs_23559BB032OutputsOutputs_FC2FACAD32"}
{attribute addProperty CRC "2239253287"}
{attribute addProperty Size "64"}
TYPE Modules_85784B27 :
STRUCT
	{attribute addProperty Name "Inputs"}
	Inputs  : Inputs_23559BB0;
	{attribute addProperty Name "Outputs"}
	Outputs  : Outputs_FC2FACAD;
END_STRUCT
END_TYPE

// ---- DUTs/IO/PDOs/Channel_830843C1.TcDUT
{attribute 'GeneratedUsingTerminal: EPP1809-0021-0016'}
{attribute addProperty BoxType "EPP1809-0021-0016"}
{attribute addProperty Id "InputAT %I*BOOL1"}
{attribute addProperty CRC "2198356929"}
{attribute addProperty Size "1"}
TYPE Channel_830843C1 EXTENDS TcoIo.InputBase_8311D824 :
STRUCT
	{attribute addProperty Name "Input"}
	Input AT %I* : BOOL;
END_STRUCT
END_TYPE

// ---- DUTs/IO/PDOs/Channel_42CA91F7.TcDUT
{attribute 'GeneratedUsingTerminal: EL2809-0015-0016'}
{attribute addProperty BoxType "EL2809-0015-0016"}
{attribute addProperty Id "OutputAT %Q*BOOL1"}
{attribute addProperty CRC "1120571895"}
{attribute addProperty Size "1"}
TYPE Channel_42CA91F7 EXTENDS TcoIo.OutputBase_10CEE7DE :
STRUCT
	{attribute addProperty Name "Output"}
	Output AT %Q* : BOOL;
END_STRUCT
END_TYPE

// ---- DUTs/IO/Boxes/EK1200_013D0B49.TcDUT
{attribute 'GeneratedUsingTerminal: EK1200-1388-0000'}
{attribute addProperty VendorId "#x00000002"}
{attribute addProperty BoxType "EK1200-1388-0000"}
{attribute addProperty Description "EK1200-5000 EtherCAT Power supply (2A E-Bus)"}
{attribute addProperty Physics "YK"}
{attribute addProperty Id "EK1200"}
{attribute addProperty CRC "20777801"}
{attribute addProperty Size "0"}
TYPE EK1200_013D0B49 EXTENDS TcoIo.EtcSlaveBoxBase_77A0E4A7 :
STRUCT
END_STRUCT
END_TYPE

// ---- DUTs/IO/Boxes/EK1122_1FC0878B.TcDUT
{attribute 'GeneratedUsingTerminal: EK1122-0000-0018'}
{attribute addProperty VendorId "#x00000002"}
{attribute addProperty BoxType "EK1122-0000-0018"}
{attribute addProperty Description "EK1122 2 port EtherCAT junction"}
{attribute addProperty Physics "KYKY"}
{attribute addProperty Id "InfoDataAT %I*InfoData_6F19DB2B2"}
{attribute addProperty CRC "532711307"}
{attribute addProperty Size "2"}
TYPE EK1122_1FC0878B EXTENDS TcoIo.EtcSlaveTerminalBase_947E5A46 :
STRUCT
	{attribute addProperty Name "InfoData"}
	InfoData : TcoIo.InfoData_6F19DB2B;
END_STRUCT
END_TYPE

// ---- DUTs/IO/Boxes/AES_510494FB.TcDUT
{attribute 'GeneratedUsingTerminal: AES-D-BC-ECAT Gen2-0001'}
{attribute addProperty VendorId "#x000001b2"}
{attribute addProperty BoxType "AES-D-BC-ECAT Gen2-0001"}
{attribute addProperty Description "AES Fieldbus Coupler Gen2"}
{attribute addProperty Physics "YY"}
{attribute addProperty Id "ModulesModules_85784B2764Device_StateAT %I*Device_State_F0482DC316Device_ControlAT %Q*Device_Control_6258066A4WcStateAT %I*WcState_9091E0EB2InfoDataAT %I*InfoData_23CBA8372"}
{attribute addProperty CRC "1359254779"}
{attribute addProperty Size "88"}
TYPE AES_510494FB EXTENDS TcoIo.EtcSlaveBoxBase_77A0E4A7 :
STRUCT
	{attribute addProperty Name "Modules"}
	Modules : Modules_85784B27;
	{attribute addProperty Name "Device_State"}
	Device_State : Device_State_F0482DC3;
	{attribute addProperty Name "Device_Control"}
	Device_Control : Device_Control_6258066A;
	{attribute addProperty Name "WcState"}
	WcState : TcoIo.WcState_9091E0EB;
	{attribute addProperty Name "InfoData"}
	InfoData : TcoIo.InfoData_23CBA837;
END_STRUCT
END_TYPE

// ---- DUTs/IO/Boxes/EPP1322_1FC0878B.TcDUT
{attribute 'GeneratedUsingTerminal: EPP1322-0001-0017'}
{attribute addProperty VendorId "#x00000002"}
{attribute addProperty BoxType "EPP1322-0001-0017"}
{attribute addProperty Description "EPP1322-0001 3 port EtherCAT P gateway"}
{attribute addProperty Physics "YYYY"}
{attribute addProperty Id "InfoDataAT %I*InfoData_6F19DB2B2"}
{attribute addProperty CRC "532711307"}
{attribute addProperty Size "2"}
TYPE EPP1322_1FC0878B EXTENDS TcoIo.EtcSlaveBoxBase_77A0E4A7 :
STRUCT
	{attribute addProperty Name "InfoData"}
	InfoData : TcoIo.InfoData_6F19DB2B;
END_STRUCT
END_TYPE

// ---- DUTs/IO/Boxes/EPP1809_32157CFD.TcDUT
{attribute 'GeneratedUsingTerminal: EPP1809-0021-0016'}
{attribute addProperty VendorId "#x00000002"}
{attribute addProperty BoxType "EPP1809-0021-0016"}
{attribute addProperty Description "EPP1809-0021 16 Ch. Dig. Input 24V, 3ms, M8"}
{attribute addProperty Physics "YY"}
{attribute addProperty Id "Channel_1AT %I*Channel_830843C11Channel_2AT %I*Channel_830843C11Channel_3AT %I*Channel_830843C11Channel_4AT %I*Channel_830843C11Channel_5AT %I*Channel_830843C11Channel_6AT %I*Channel_830843C11Channel_7AT %I*Channel_830843C11Channel_8AT %I*Channel_830843C11Channel_9AT %I*Channel_830843C11Channel_10AT %I*Channel_830843C11Channel_11AT %I*Channel_830843C11Channel_12AT %I*Channel_830843C11Channel_13AT %I*Channel_830843C11Channel_14AT %I*Channel_830843C11Channel_15AT %I*Channel_830843C11Channel_16AT %I*Channel_830843C11WcStateAT %I*WcState_9091E0EB2InfoDataAT %I*InfoData_6F19DB2B2"}
{attribute addProperty CRC "840269053"}
{attribute addProperty Size "20"}
TYPE EPP1809_32157CFD EXTENDS TcoIo.EtcSlaveBoxBase_77A0E4A7 :
STRUCT
	{attribute addProperty Name "Channel_1"}
	Channel_1 : Channel_830843C1;
	{attribute addProperty Name "Channel_2"}
	Channel_2 : Channel_830843C1;
	{attribute addProperty Name "Channel_3"}
	Channel_3 : Channel_830843C1;
	{attribute addProperty Name "Channel_4"}
	Channel_4 : Channel_830843C1;
	{attribute addProperty Name "Channel_5"}
	Channel_5 : Channel_830843C1;
	{attribute addProperty Name "Channel_6"}
	Channel_6 : Channel_830843C1;
	{attribute addProperty Name "Channel_7"}
	Channel_7 : Channel_830843C1;
	{attribute addProperty Name "Channel_8"}
	Channel_8 : Channel_830843C1;
	{attribute addProperty Name "Channel_9"}
	Channel_9 : Channel_830843C1;
	{attribute addProperty Name "Channel_10"}
	Channel_10 : Channel_830843C1;
	{attribute addProperty Name "Channel_11"}
	Channel_11 : Channel_830843C1;
	{attribute addProperty Name "Channel_12"}
	Channel_12 : Channel_830843C1;
	{attribute addProperty Name "Channel_13"}
	Channel_13 : Channel_830843C1;
	{attribute addProperty Name "Channel_14"}
	Channel_14 : Channel_830843C1;
	{attribute addProperty Name "Channel_15"}
	Channel_15 : Channel_830843C1;
	{attribute addProperty Name "Channel_16"}
	Channel_16 : Channel_830843C1;
	{attribute addProperty Name "WcState"}
	WcState : TcoIo.WcState_9091E0EB;
	{attribute addProperty Name "InfoData"}
	InfoData : TcoIo.InfoData_6F19DB2B;
END_STRUCT
END_TYPE

// ---- DUTs/IO/Boxes/EPP1008_78E8D3DD.TcDUT
{attribute 'GeneratedUsingTerminal: EPP1008-0001-0017'}
{attribute addProperty VendorId "#x00000002"}
{attribute addProperty BoxType "EPP1008-0001-0017"}
{attribute addProperty Description "EPP1008-0001 8 Ch. Dig. Input 24V, 3ms, M8"}
{attribute addProperty Physics "YY"}
{attribute addProperty Id "Channel_1AT %I*Channel_830843C11Channel_2AT %I*Channel_830843C11Channel_3AT %I*Channel_830843C11Channel_4AT %I*Channel_830843C11Channel_5AT %I*Channel_830843C11Channel_6AT %I*Channel_830843C11Channel_7AT %I*Channel_830843C11Channel_8AT %I*Channel_830843C11WcStateAT %I*WcState_9091E0EB2InfoDataAT %I*InfoData_6F19DB2B2"}
{attribute addProperty CRC "2028524509"}
{attribute addProperty Size "12"}
TYPE EPP1008_78E8D3DD EXTENDS TcoIo.EtcSlaveBoxBase_77A0E4A7 :
STRUCT
	{attribute addProperty Name "Channel_1"}
	Channel_1 : Channel_830843C1;
	{attribute addProperty Name "Channel_2"}
	Channel_2 : Channel_830843C1;
	{attribute addProperty Name "Channel_3"}
	Channel_3 : Channel_830843C1;
	{attribute addProperty Name "Channel_4"}
	Channel_4 : Channel_830843C1;
	{attribute addProperty Name "Channel_5"}
	Channel_5 : Channel_830843C1;
	{attribute addProperty Name "Channel_6"}
	Channel_6 : Channel_830843C1;
	{attribute addProperty Name "Channel_7"}
	Channel_7 : Channel_830843C1;
	{attribute addProperty Name "Channel_8"}
	Channel_8 : Channel_830843C1;
	{attribute addProperty Name "WcState"}
	WcState : TcoIo.WcState_9091E0EB;
	{attribute addProperty Name "InfoData"}
	InfoData : TcoIo.InfoData_6F19DB2B;
END_STRUCT
END_TYPE

// ---- DUTs/IO/Boxes/EL1809_32157CFD.TcDUT
{attribute 'GeneratedUsingTerminal: EL1809-0000-0018'}
{attribute addProperty VendorId "#x00000002"}
{attribute addProperty BoxType "EL1809-0000-0018"}
{attribute addProperty Description "EL1809 16Ch. Dig. Input 24V, 3ms"}
{attribute addProperty Physics "KK"}
{attribute addProperty Id "Channel_1AT %I*Channel_830843C11Channel_2AT %I*Channel_830843C11Channel_3AT %I*Channel_830843C11Channel_4AT %I*Channel_830843C11Channel_5AT %I*Channel_830843C11Channel_6AT %I*Channel_830843C11Channel_7AT %I*Channel_830843C11Channel_8AT %I*Channel_830843C11Channel_9AT %I*Channel_830843C11Channel_10AT %I*Channel_830843C11Channel_11AT %I*Channel_830843C11Channel_12AT %I*Channel_830843C11Channel_13AT %I*Channel_830843C11Channel_14AT %I*Channel_830843C11Channel_15AT %I*Channel_830843C11Channel_16AT %I*Channel_830843C11WcStateAT %I*WcState_9091E0EB2InfoDataAT %I*InfoData_6F19DB2B2"}
{attribute addProperty CRC "840269053"}
{attribute addProperty Size "20"}
TYPE EL1809_32157CFD EXTENDS TcoIo.EtcSlaveTerminalBase_947E5A46 :
STRUCT
	{attribute addProperty Name "Channel_1"}
	Channel_1 : Channel_830843C1;
	{attribute addProperty Name "Channel_2"}
	Channel_2 : Channel_830843C1;
	{attribute addProperty Name "Channel_3"}
	Channel_3 : Channel_830843C1;
	{attribute addProperty Name "Channel_4"}
	Channel_4 : Channel_830843C1;
	{attribute addProperty Name "Channel_5"}
	Channel_5 : Channel_830843C1;
	{attribute addProperty Name "Channel_6"}
	Channel_6 : Channel_830843C1;
	{attribute addProperty Name "Channel_7"}
	Channel_7 : Channel_830843C1;
	{attribute addProperty Name "Channel_8"}
	Channel_8 : Channel_830843C1;
	{attribute addProperty Name "Channel_9"}
	Channel_9 : Channel_830843C1;
	{attribute addProperty Name "Channel_10"}
	Channel_10 : Channel_830843C1;
	{attribute addProperty Name "Channel_11"}
	Channel_11 : Channel_830843C1;
	{attribute addProperty Name "Channel_12"}
	Channel_12 : Channel_830843C1;
	{attribute addProperty Name "Channel_13"}
	Channel_13 : Channel_830843C1;
	{attribute addProperty Name "Channel_14"}
	Channel_14 : Channel_830843C1;
	{attribute addProperty Name "Channel_15"}
	Channel_15 : Channel_830843C1;
	{attribute addProperty Name "Channel_16"}
	Channel_16 : Channel_830843C1;
	{attribute addProperty Name "WcState"}
	WcState : TcoIo.WcState_9091E0EB;
	{attribute addProperty Name "InfoData"}
	InfoData : TcoIo.InfoData_6F19DB2B;
END_STRUCT
END_TYPE

// ---- DUTs/IO/Boxes/EL2809_2B6483BD.TcDUT
{attribute 'GeneratedUsingTerminal: EL2809-0015-0016'}
{attribute addProperty VendorId "#x00000002"}
{attribute addProperty BoxType "EL2809-0015-0016"}
{attribute addProperty Description "EL2809-0015 16Ch. Dig. Output 24V DC, 0.35A, not short-circuit proof"}
{attribute addProperty Physics "KK"}
{attribute addProperty Id "Channel_1AT %Q*Channel_42CA91F71Channel_2AT %Q*Channel_42CA91F71Channel_3AT %Q*Channel_42CA91F71Channel_4AT %Q*Channel_42CA91F71Channel_5AT %Q*Channel_42CA91F71Channel_6AT %Q*Channel_42CA91F71Channel_7AT %Q*Channel_42CA91F71Channel_8AT %Q*Channel_42CA91F71Channel_9AT %Q*Channel_42CA91F71Channel_10AT %Q*Channel_42CA91F71Channel_11AT %Q*Channel_42CA91F71Channel_12AT %Q*Channel_42CA91F71Channel_13AT %Q*Channel_42CA91F71Channel_14AT %Q*Channel_42CA91F71Channel_15AT %Q*Channel_42CA91F71Channel_16AT %Q*Channel_42CA91F71WcStateAT %I*WcState_0B2B16F91InfoDataAT %I*InfoData_6F19DB2B2"}
{attribute addProperty CRC "728007613"}
{attribute addProperty Size "19"}
TYPE EL2809_2B6483BD EXTENDS TcoIo.EtcSlaveTerminalBase_947E5A46 :
STRUCT
	{attribute addProperty Name "Channel_1"}
	Channel_1 : Channel_42CA91F7;
	{attribute addProperty Name "Channel_2"}
	Channel_2 : Channel_42CA91F7;
	{attribute addProperty Name "Channel_3"}
	Channel_3 : Channel_42CA91F7;
	{attribute addProperty Name "Channel_4"}
	Channel_4 : Channel_42CA91F7;
	{attribute addProperty Name "Channel_5"}
	Channel_5 : Channel_42CA91F7;
	{attribute addProperty Name "Channel_6"}
	Channel_6 : Channel_42CA91F7;
	{attribute addProperty Name "Channel_7"}
	Channel_7 : Channel_42CA91F7;
	{attribute addProperty Name "Channel_8"}
	Channel_8 : Channel_42CA91F7;
	{attribute addProperty Name "Channel_9"}
	Channel_9 : Channel_42CA91F7;
	{attribute addProperty Name "Channel_10"}
	Channel_10 : Channel_42CA91F7;
	{attribute addProperty Name "Channel_11"}
	Channel_11 : Channel_42CA91F7;
	{attribute addProperty Name "Channel_12"}
	Channel_12 : Channel_42CA91F7;
	{attribute addProperty Name "Channel_13"}
	Channel_13 : Channel_42CA91F7;
	{attribute addProperty Name "Channel_14"}
	Channel_14 : Channel_42CA91F7;
	{attribute addProperty Name "Channel_15"}
	Channel_15 : Channel_42CA91F7;
	{attribute addProperty Name "Channel_16"}
	Channel_16 : Channel_42CA91F7;
	{attribute addProperty Name "WcState"}
	WcState : TcoIo.WcState_0B2B16F9;
	{attribute addProperty Name "InfoData"}
	InfoData : TcoIo.InfoData_6F19DB2B;
END_STRUCT
END_TYPE

// ---- DUTs/IO/Boxes/EL9011_D65D3D32.TcDUT
{attribute 'GeneratedUsingTerminal: EL9011--0000'}
{attribute addProperty VendorId "#x00000002"}
{attribute addProperty BoxType "EL9011--0000"}
{attribute addProperty Description "EL9011 End Terminal"}
{attribute addProperty Physics ""}
{attribute addProperty Id "EL9011"}
{attribute addProperty CRC "3596434738"}
{attribute addProperty Size "0"}
TYPE EL9011_D65D3D32 EXTENDS TcoIo.EtcSlaveEndTerminalBase_866C7F0C :
STRUCT
END_STRUCT
END_TYPE

// ---- DUTs/IO/Devices/SyncUnitTasks_4BE01469.TcDUT
{attribute 'GeneratedUsingTerminal: '}
{attribute addProperty BoxType ""}
{attribute addProperty Id "unreferencedAT %I*SyncUnitTask_AB2F50799PlcTaskAT %I*SyncUnitTask_AB2F50799"}
{attribute addProperty CRC "1272976489"}
{attribute addProperty Size "18"}
TYPE SyncUnitTasks_4BE01469 EXTENDS TcoIo.SyncUnitTasksBase_7C8711EB :
STRUCT
	{attribute addProperty Name "unreferenced"}
	unreferenced : TcoIo.SyncUnitTask_AB2F5079;
	{attribute addProperty Name "PlcTask"}
	PlcTask : TcoIo.SyncUnitTask_AB2F5079;
END_STRUCT
END_TYPE

// ---- DUTs/IO/Devices/SyncUnits_67D36DDA.TcDUT
{attribute 'GeneratedUsingTerminal: '}
{attribute addProperty BoxType ""}
{attribute addProperty Id "_defaultAT %I*SyncUnitTasks_4BE0146918"}
{attribute addProperty CRC "1741909466"}
{attribute addProperty Size "18"}
TYPE SyncUnits_67D36DDA EXTENDS TcoIo.SyncUnitsBase_AD6C35CE :
STRUCT
	{attribute addProperty Name "_default"}
	_default : SyncUnitTasks_4BE01469;
END_STRUCT
END_TYPE

// ---- DUTs/IO/Topology/EK_E812B8FA.TcDUT
{attribute 'GeneratedUsingTerminal: EK1122-0000-0018'}
{attribute addProperty BoxType "EK1122-0000-0018"}
{attribute addProperty Id "PNEUAES_510494FB88ABEPP1322_1FC0878B2AB21EPP1809_32157CFD20AB22EPP1809_32157CFD20AB23EPP1008_78E8D3DD12AB24EPP1008_78E8D3DD12"}
{attribute addProperty CRC "3893541114"}
{attribute addProperty Size "154"}
{attribute addProperty Name "EK"}
TYPE EK_E812B8FA EXTENDS EK1122_1FC0878B :
STRUCT
	{attribute addProperty Name "PNEU"}
	{attribute addProperty PreviousPort "EK : D"}
	{attribute addProperty SyncUnit "default"}
	PNEU : AES_510494FB;
	{attribute addProperty Name "AB"}
	{attribute addProperty PreviousPort "PNEU : B"}
	{attribute addProperty SyncUnit "default"}
	AB : EPP1322_1FC0878B;
	{attribute addProperty Name "AB21"}
	{attribute addProperty PreviousPort "AB : C"}
	{attribute addProperty SyncUnit "default"}
	AB21 : EPP1809_32157CFD;
	{attribute addProperty Name "AB22"}
	{attribute addProperty PreviousPort "AB21 : B"}
	{attribute addProperty SyncUnit "default"}
	AB22 : EPP1809_32157CFD;
	{attribute addProperty Name "AB23"}
	{attribute addProperty PreviousPort "AB22 : B"}
	{attribute addProperty SyncUnit "default"}
	AB23 : EPP1008_78E8D3DD;
	{attribute addProperty Name "AB24"}
	{attribute addProperty PreviousPort "AB23 : B"}
	{attribute addProperty SyncUnit "default"}
	AB24 : EPP1008_78E8D3DD;
END_STRUCT
END_TYPE

// ---- DUTs/IO/Topology/EC_4E5C738F.TcDUT
{attribute 'GeneratedUsingTerminal: EK1200-1388-0000'}
{attribute addProperty BoxType "EK1200-1388-0000"}
{attribute addProperty Id "EKEK_E812B8FA154IA1EL1809_32157CFD20QA1EL2809_2B6483BD19Term_11_EL9011EL9011_D65D3D320"}
{attribute addProperty CRC "1314681743"}
{attribute addProperty Size "193"}
{attribute addProperty Name "EC"}
TYPE EC_4E5C738F EXTENDS EK1200_013D0B49 :
STRUCT
	{attribute addProperty Name "EK"}
	{attribute addProperty PreviousPort "EC : B"}
	{attribute addProperty SyncUnit "default"}
	EK : EK_E812B8FA;
	{attribute addProperty Name "IA1"}
	{attribute addProperty PreviousPort "EK : C"}
	{attribute addProperty SyncUnit "default"}
	IA1 : EL1809_32157CFD;
	{attribute addProperty Name "QA1"}
	{attribute addProperty PreviousPort "IA1 : B"}
	{attribute addProperty SyncUnit "default"}
	QA1 : EL2809_2B6483BD;
	{attribute addProperty Name "Term 11 (EL9011)"}
	{attribute addProperty PreviousPort "QA1 : B"}
	{attribute addProperty SyncUnit "default"}
	Term_11_EL9011 : EL9011_D65D3D32;
END_STRUCT
END_TYPE

// ---- DUTs/IO/Topology/EC_245FBB9A.TcDUT
{attribute 'GeneratedUsingTerminal: IODEVICETYPE_ETHERCATPROT'}
{attribute addProperty BoxType "IODEVICETYPE_ETHERCATPROT"}
{attribute addProperty Id "ECEC_4E5C738F193SyncUnitsSyncUnits_67D36DDA18InputsInputs_A65FACA410OutputsOutputs_23C0ED1D6InfoDataInfoData_84133AC922"}
{attribute addProperty CRC "610253722"}
{attribute addProperty Size "249"}
{attribute addProperty Name "EC"}
TYPE EC_245FBB9A EXTENDS TcoIo.EtcMasterBase_62654B43 :
STRUCT
	{attribute addProperty Name "EC"}
	{attribute addProperty PreviousPort "EC : Master"}
	{attribute addProperty SyncUnit "default"}
	EC : EC_4E5C738F;
	{attribute addProperty Name "SyncUnits"}
	SyncUnits : SyncUnits_67D36DDA;
	{attribute addProperty Name "Inputs"}
	Inputs : TcoIo.Inputs_A65FACA4;
	{attribute addProperty Name "Outputs"}
	Outputs : TcoIo.Outputs_23C0ED1D;
	{attribute addProperty Name "InfoData"}
	InfoData : TcoIo.InfoData_84133AC9;
END_STRUCT
END_TYPE

// ---- GVLs/GVL_iXlinker.TcGVL
{attribute 'qualified_only'}
VAR_GLOBAL
		EC : EC_245FBB9A;
		IN : EL1809_32157CFD;
		OUT : EL2809_2B6483BD;
		{attribute addProperty Name "B10.1"} 
		B10_1 : BOOL;
		
		B20_1 : BOOL;
END_VAR

// B10

// ---- Abstractions/CUBase/ICUBase.TcIO
INTERFACE ICUBase

PROPERTY AutomatTask : REFERENCE TO CUBaseAutomat
GET
END_GET
END_PROPERTY

PROPERTY GroundTask : REFERENCE TO CUBaseGround
GET
END_GET
END_PROPERTY

PROPERTY  ManualTask : REFERENCE TO TcoTaskedService
GET
END_GET
END_PROPERTY

PROPERTY ProcessDataManager : REFERENCE TO ProcessDataManager
GET
END_GET
END_PROPERTY

PROPERTY RecoverTask : REFERENCE TO CUBaseRecover
GET
END_GET
END_PROPERTY

PROPERTY StatusInfo :REFERENCE TO CuBaseStatusInfo
GET
END_GET
END_PROPERTY

PROPERTY SuspendTask : REFERENCE TO CUBaseSuspend
GET
END_GET
END_PROPERTY

END_INTERFACE

// ---- Abstractions/CUBase/ICUTask.TcIO
INTERFACE ICUTask

PROPERTY Task : REFERENCE TO TcoCore.TcoTask
GET
END_GET
END_PROPERTY

END_INTERFACE

// ---- Abstractions/Safety/ControlButtons/ITcoControlButtons.TcIO
INTERFACE ITcoControlButtons

PROPERTY ButtonAuto : BOOL
GET
END_GET
SET
END_SET
END_PROPERTY

PROPERTY ButtonGround : BOOL
GET
END_GET
SET
END_SET
END_PROPERTY

PROPERTY ButtonRecover : BOOL
GET
END_GET
SET
END_SET
END_PROPERTY

PROPERTY ButtonSuspend : BOOL
GET
END_GET
SET
END_SET
END_PROPERTY

END_INTERFACE

// ---- Abstractions/Safety/ControlVoltage/ITcoControlVoltage.TcIO
INTERFACE ITcoControlVoltage

PROPERTY IsOff : BOOL
GET
END_GET
END_PROPERTY

PROPERTY IsOn : BOOL
GET
END_GET
END_PROPERTY

END_INTERFACE

// ---- Abstractions/Safety/DoorCircuit/ITcoDoorCircuit.TcIO
INTERFACE ITcoDoorCircuit

{attribute 'monitoring' := 'call'}
PROPERTY IsClosed : BOOL
GET
END_GET
END_PROPERTY

{attribute 'monitoring' := 'call'}
PROPERTY IsGlobalVoltageOk : BOOL
GET
END_GET
END_PROPERTY

{attribute 'monitoring' := 'call'}
PROPERTY IsLocalDoorsVoltageOk : BOOL
GET
END_GET
END_PROPERTY

{attribute 'monitoring' := 'call'}
PROPERTY IsLocalVoltageOk : BOOL
GET
END_GET
END_PROPERTY

{attribute 'monitoring' := 'call'}
PROPERTY IsLocked : BOOL
GET
END_GET
END_PROPERTY

{attribute 'monitoring' := 'call'}
PROPERTY IsUnLocked : BOOL
GET
END_GET
END_PROPERTY

METHOD Lock : BOOL
VAR_INPUT
END_VAR
END_METHOD

METHOD UnLock : BOOL
VAR_INPUT
END_VAR
END_METHOD

END_INTERFACE

// ---- Abstractions/Safety/Doors/ITcoDoorLock.TcIO
INTERFACE ITcoDoorLock

{attribute 'monitoring' := 'call'}
PROPERTY IsClosed : BOOL
GET
END_GET
END_PROPERTY

{attribute 'monitoring' := 'call'}
PROPERTY IsLocked : BOOL
GET
END_GET
END_PROPERTY

{attribute 'monitoring' := 'call'}
PROPERTY IsOpen : BOOL
GET
END_GET
END_PROPERTY

METHOD Lock : BOOL
VAR_INPUT
END_VAR
END_METHOD

METHOD UnLock : BOOL
VAR_INPUT
END_VAR
END_METHOD

END_INTERFACE

// ---- Abstractions/Safety/KeyMode/ITcoKeyMode.TcIO
INTERFACE ITcoKeyMode

PROPERTY KeyInAuto : BOOL
GET
END_GET
END_PROPERTY

PROPERTY KeyInManual : BOOL
GET
END_GET
END_PROPERTY

PROPERTY KeyInStep : BOOL
GET
END_GET
END_PROPERTY

END_INTERFACE

// ---- Abstractions/Safety/KeyNormalService/ITcoKeyNormalSevice.TcIO
INTERFACE ITcoKeyNormalSevice

PROPERTY KeyInNormal : BOOL
GET
END_GET
END_PROPERTY

PROPERTY KeyInService : BOOL
GET
END_GET
END_PROPERTY

END_INTERFACE

// ---- MAIN.TcPOU
PROGRAM MAIN
VAR
    _technology : Technology;
END_VAR

_technology.Run();

END_PROGRAM

// ---- Technology/Technology.TcPOU
FUNCTION_BLOCK Technology EXTENDS TcoCore.TcoContext
VAR	
    _processSettings     : ProcessDataManager(THIS^);  			//a.k.a receipe
	_reworkSettings     : ProcessDataManager(THIS^);  			//a.k.a receipe for rework
    _technologySettings  : TechnologicalDataManager(THIS^);		//a.k.a machine settings
    _processTraceability : ProcessDataManager(THIS^);			//the same structure as process setting but filled with actual production data (measurements, inspection results, etc)
	
	
	fbGetCurTaskIndex            : GETCURTASKINDEX;
	_notificationPanel      : NotificationPanel(THIS^);				//provide technology state signals to side baner in visualisation
    {attribute addProperty Name "<#AUTOMAT ALL#>"}
    _automatAllTask : TcoCore.TcoTask(THIS^);					// Commmand-like taks to execute automation mode on whole technology. Handled in controlled units.
    {attribute addProperty Name "<#GROUND ALL#>"}
    _groundAllTask : TcoCore.TcoTask(THIS^);	

	{attribute addProperty Name "<#_cu00x#>"}					
    _cu00x         : CU00x(THIS^);
	
	{attribute addProperty Name "<#Technology Components#>"}	
	_components : TechnologyComponents:= (Parent := THIS^);

	{attribute addProperty Name "Device 1 (EtherCAT)"}
	Device_1 : TcoIo.TcoEthercatMasterDevice(THIS^);
	
	_setDummyConditionsSuffisient:BOOL;
	_dummyBlinker              : TcoUtilities.TcoBlinker(THIS^);
END_VAR

METHOD AllowAutomat : BOOL
VAR_INPUT
END_VAR
AllowAutomat := TRUE;
END_METHOD

METHOD AllowGround : BOOL
VAR_INPUT
END_VAR
AllowGround := TRUE;
END_METHOD

METHOD AllowManual :  BOOL
VAR_INPUT
END_VAR
AllowManual := TRUE;
END_METHOD

PROPERTY AutomatAllTask : REFERENCE TO TcoCore.TcoTask
GET
AutomatAllTask REF= _automatAllTask;
END_GET
END_PROPERTY

PROPERTY PUBLIC Cu00x : Reference to CU00x
GET
Cu00x REF=_cu00x;
END_GET
END_PROPERTY

METHOD ForceStepMode : BOOL
ForceStepMode := FALSE;
END_METHOD

PROPERTY GroundAllTask : REFERENCE TO TcoCore.TcoTask
GET
GroundAllTask REF= _groundAllTask;
END_GET
END_PROPERTY

METHOD InitializeComponents
VAR_INPUT
END_VAR

VAR
	controlVolage: BOOL;
	controlVoltageDoor: BOOL;
	estop: BOOL;
	presure: BOOL;
	locked: BOOL;
	lock: BOOL;
	opened: BOOL;
	closed: BOOL;
	
END_VAR
controlVolage:=FALSE;
controlVoltageDoor:=FALSE;
estop:=FALSE;
presure:=FALSE;

//_dummyBlinker(inOffTime := T#10000MS, inOnTime := T#10000MS);
(*
closed:=GVL_iXlinker.EC1.EK1200.IA1_EL1809.Channel_8.Input;
locked:=GVL_iXlinker.EC1.EK1200.IA1_EL1809.Channel_9.Input;

IF _setDummyConditionsSuffisient THEN
	controlVolage:=TRUE;
	controlVoltageDoor:=TRUE;
	estop:=FALSE;
	presure:=TRUE;


END_IF;

_components.ModeKey(inoKeyState1:=GVL_iXlinker.EC1.EK1200.IA1_EL1809.Channel_1.Input ,
					inoKeyState2:=GVL_iXlinker.EC1.EK1200.IA1_EL1809.Channel_2.Input);
					
_components.NormalServiceKey(inoSignal:=GVL_iXlinker.EC1.EK1200.IA1_EL1809.Channel_3.Input);
					
_components.ControlButtons(
	inoButtonRecover:=GVL_iXlinker.EC1.EK1200.IA1_EL1809.Channel_4.Input  , 
	inoButtonSuspend:=GVL_iXlinker.EC1.EK1200.IA1_EL1809.Channel_5.Input  , 
	inoButtonGround:=GVL_iXlinker.EC1.EK1200.IA1_EL1809.Channel_6.Input , 
	inoButtonAuto:=GVL_iXlinker.EC1.EK1200.IA1_EL1809.Channel_7.Input, 
	inoButtonRecoverLight:=GVL_iXlinker.EC1.EK1200.QA1_EL2809.Channel_1.Output  , 
	inoButtonSuspendLight:=GVL_iXlinker.EC1.EK1200.QA1_EL2809.Channel_2.Output  , 
	inoButtonGroundLight:=GVL_iXlinker.EC1.EK1200.QA1_EL2809.Channel_3.Output  , 
	inoButtonAutoLight:= GVL_iXlinker.EC1.EK1200.QA1_EL2809.Channel_4.Output );
	

					

_components.GlobalControlVoltage(inoSignal := controlVolage);

_components.LocalControlVoltage(inoSignal := controlVolage);
_components.LocalDoorVoltage(inoSignal := controlVoltageDoor);

_components.EmergencyStop(inoSignal := estop);
_components.AirPresureOk(inoSignal:= presure);


_components.StandardDoor(inoIsLocked := locked,
    inoIsOpen := opened,
    inoLock :=lock);
	
	
_components.BasicDoor(inoIsClosed := closed,
     inoLock := lock);


_components.DoorCicuit();

_components.Zone(inDoorCircuit:=_components.DoorCicuit,
				inEstopActive:=_components.EmergencyStop.Signal,
				inAirPressureOK:= _components.AirPresureOk.Signal);
		
				
_components.Zone.Service();
*)
END_METHOD

METHOD InitializeComponentsOnce
VAR_INPUT
END_VAR
_components.DoorCicuit.Restore();
_components.Zone.Restore();



_components.DoorCicuit.AddDoors(inDoor:=_components.StandardDoor);
_components.DoorCicuit.AddDoors(inDoor:=_components.BasicDoor);
_components.DoorCicuit.AddGlobalVoltage(inVoltage:=_components.GlobalControlVoltage);
_components.DoorCicuit.AddLocalVoltage(inVoltage:=_components.LocalControlVoltage);
_components.DoorCicuit.AddLocalDoorsVoltage(inVoltage:=_components.LocalDoorVoltage);


_components.Zone.AddControlledUnit(inControlledUnit:=_cu00x);
_components.Zone.AddControlButtons(inControlButtons:=_components.ControlButtons);
_components.Zone.AddKeyMode(inKeyMode:=_components.ModeKey);
_components.Zone.AddKeyNormalService(inKeyNormalService:=_components.NormalServiceKey);
END_METHOD

(*~
	<docu>
		<summary>
			Main method of the TcoContext. This is the entry point of any control logic that belongs to this context. 
			The call of this method is ensured by calling the <c>InstanceName.Run()</c> method, and it must not be called explicitly.
			This method is abstract, and it must be overridden in derived block.
		</summary>
	</docu>
~*)
METHOD PROTECTED Main
VAR
	_notificationSourceSignals: NotificationPanelInfo;
	safetyCircuitOk: BOOL;
	_eStopActive: BOOL;
	_keysAto: BOOL;
	_closed: BOOL;
	_locked: BOOL;
END_VAR
(*
	Context settings 
*)

// RTC Synchronisation
THIS^.RtcSynchronize(TRUE,  
					 '192.168.4.1.1.1',    // Provide AMS ID of the time source, leave blank if local. 
					 60);

// Messenger logger settings
_settings.Messaging.MessageDigestMethod := eMessageDigestMethod.CRC32;
_settings.Messaging.MessengerLoggingMethod := eMessengerLogMethod.OnEventRisen;


_components.DoorCicuit.Config.MaxDoors:=12;
_components.DoorCicuit.Config.MaxGlobalVoltage:=2;
_components.DoorCicuit.Config.MaxLocalVoltage:=2;
_components.DoorCicuit.Config.MaxLocalDoorsVoltage:=2;


_components.Zone.Config.MaxControlButtons:=2;
_components.Zone.Config.MaxControledUnits:=10;
_components.Zone.Config.MaxKeyMode:=2;
_components.Zone.Config.MaxKeyNormalService:=2;



THIS^.InitializeComponents();
fbGetCurTaskIndex();
IF _TaskInfo[fbGetCurTaskIndex.index].FirstCycle THEN
    // The code that you want to be executed at the first cycle of  PLC only 
	THIS^.InitializeComponentsOnce();
END_IF

//notification panel
 Context.Environment.Messaging.Suspend();
			
_closed:=TRUE;
//_closed   := 	Components.Safety.DoorCircuits.DoorCircuit_2.IsClosed 
//			AND Components.Safety.DoorCircuits.DoorCircuit_3.IsClosed  
//			AND Components.Safety.DoorCircuits.DoorCircuit_4.IsClosed  
//			AND Components.Safety.DoorCircuits.DoorCircuit_5.IsClosed  
//			AND Components.Safety.DoorCircuits.DoorCircuit_6.IsClosed;

 _locked:=TRUE;
//_locked   := 	Components.Safety.DoorCircuits.DoorCircuit_2.IsLocked 
//			AND Components.Safety.DoorCircuits.DoorCircuit_3.IsLocked  
//			AND Components.Safety.DoorCircuits.DoorCircuit_4.IsLocked  
//			AND Components.Safety.DoorCircuits.DoorCircuit_5.IsLocked  
//			AND Components.Safety.DoorCircuits.DoorCircuit_6.IsLocked;
			
_keysAto  := TRUE;
_eStopActive:=0;


_notificationSourceSignals.ControlVoltage   := TRUE;//Components.ControlVoltage.Signal.Signal 
_notificationSourceSignals.AirPressure      := TRUE;//Components.AirPressureOk.Signal.Signal, 
_notificationSourceSignals.AutomatAllowed   := _keysAto; 
_notificationSourceSignals.EmergencyStop    := _eStopActive > 0; 
_notificationSourceSignals.SafetyDoorOk     :=safetyCircuitOk;	
_notificationSourceSignals.LightCurtain     := TRUE; 	// not used
_notificationSourceSignals.DoorClosed       := _closed; 
_notificationSourceSignals.DoorLocked       := _locked; 
_notificationSourceSignals.ProcessDataOk    := _processSettings._data._EntityId <> '';
_notificationSourceSignals.TechnologyDataOk := _technologySettings._data._EntityId <> '';  
	
_notificationPanel(inBlinkPeriod:=T#500MS , inSignalSource:=_notificationSourceSignals );
			
 Context.Environment.Messaging.Resume();

(*
	
	Data managers

*)

_processSettings();
_reworkSettings();
_technologySettings();

(*

	Controlled units
	
*)

_cu00x();


_automatAllTask();
_groundAllTask();

//Device_1(	SyncUnits		:= ADR(		GVL_iXlinker.EC1.SyncUnits),
//			SyncUnitsSize	:= SIZEOF(	GVL_iXlinker.EC1.SyncUnits),
//			Inputs			:=			GVL_iXlinker.EC1.Inputs,
//			InfoData		:=			GVL_iXlinker.EC1.InfoData);
END_METHOD


(*~
	<docu>
		<summary>
			Called upon exit from the context. When overridden in derived class allows to execute an arbitrary logic after closing the context cycle.	
		</summary>			
	</docu>	
~*)METHOD PROTECTED OnExit
_automatAllTask.DoneWhen(TRUE);
_groundAllTask.DoneWhen(TRUE);
END_METHOD

PROPERTY ProcessSettings : REFERENCE TO ProcessDataManager
GET
ProcessSettings REF= _processSettings;
END_GET
END_PROPERTY

PROPERTY ReworkSettings : REFERENCE TO ProcessDataManager
GET
ReworkSettings REF= _reworkSettings;
END_GET
END_PROPERTY

PROPERTY TechnologicalSettings : REFERENCE TO TechnologicalDataManager
GET
TechnologicalSettings REF= _technologySettings;
END_GET
END_PROPERTY

END_FUNCTION_BLOCK

// ---- Technology/Data/ProcessDataManager.TcPOU
FUNCTION_BLOCK ProcessDataManager EXTENDS TcoData.TcoDataExchange
VAR
    _data : ProcessData := (Parent := THIS^);
	_sb : TcoCore.StringBuilder;
END_VAR

SUPER^();

PROPERTY Data : REFERENCE TO ProcessData
GET
Data REF= _data;
END_GET
END_PROPERTY

END_FUNCTION_BLOCK

// ---- Technology/Data/TechnologicalDataManager.TcPOU
FUNCTION_BLOCK TechnologicalDataManager EXTENDS TcoData.TcoDataExchange
VAR
    _data : TechnologyData := (Parent := THIS^);
END_VAR

SUPER^();

PROPERTY Data : REFERENCE TO TechnologyData
GET
Data REF= _data;
END_GET
END_PROPERTY

END_FUNCTION_BLOCK

// ---- Abstractions/Generic/NotificationPanel/NotificationPanel.TcPOU
{attribute wpf [Container(Layout.Stack)]}
FUNCTION_BLOCK NotificationPanel EXTENDS TcoObject
VAR_INPUT
	(*~
		<docu>
			<summary>
				Time duration for toggle signal.
			</summary>
		</docu>
	~*)
	inBlinkPeriod:TIME;
		(*~
		<docu>
			<summary>
				Source inputs for signalisation.
			</summary>
		</docu>
	~*)
	inSignalSource:NotificationPanelInfo;
	
END_VAR
VAR
	{attribute addProperty Name "<#Heart beat#>"}
  	_heartBeat : BOOL;
	
    {attribute clr [RenderIgnore()]}
	_badgeValue : INT;

	{attribute clr [RenderIgnore()]}
    _toggle: TcoUtilities.TcoBlinker(THIS^);

	_notificationPanelSignals: NotificationPanelInfo;
END_VAR

_toggle(inOffTime:=inBlinkPeriod,inOnTime:=inBlinkPeriod);
_heartBeat := _toggle.IsOn;
_notificationPanelSignals:=inSignalSource;

_badgeValue := 0;
_badgeValue:=_badgeValue + BOOL_TO_INT(NOT _notificationPanelSignals.ControlVoltage);
_badgeValue:=_badgeValue + BOOL_TO_INT(NOT _notificationPanelSignals.AirPressure);
_badgeValue:=_badgeValue + BOOL_TO_INT(NOT _notificationPanelSignals.AutomatAllowed);
_badgeValue:=_badgeValue + BOOL_TO_INT(_notificationPanelSignals.EmergencyStop);
_badgeValue:=_badgeValue + BOOL_TO_INT(NOT _notificationPanelSignals.SafetyDoorOk);
_badgeValue:=_badgeValue + BOOL_TO_INT(NOT _notificationPanelSignals.DoorClosed);
_badgeValue:=_badgeValue + BOOL_TO_INT(NOT _notificationPanelSignals.Doorlocked);
_badgeValue:=_badgeValue + BOOL_TO_INT(NOT _notificationPanelSignals.LightCurtain);
_badgeValue:=_badgeValue + BOOL_TO_INT(NOT _notificationPanelSignals.ProcessDataOk);
_badgeValue:=_badgeValue + BOOL_TO_INT(NOT _notificationPanelSignals.TechnologyDataOk);

END_FUNCTION_BLOCK

// ---- Technology/CU00x/CU00x.TcPOU
{attribute addProperty ShortName "CU00x"}
{attribute addProperty Name "Controlled unit x_tempalte_x"}
FUNCTION_BLOCK CU00x EXTENDS CUBase 
VAR
    _cuProcessDataDisplay       :  CU00xProcessData := (Parent := THIS^);
    _cuTechnologicalDataDisplay :  CU00xTechnologicalData := (Parent := THIS^);
    _components          		:  CU00xComponents := (Parent := THIS^);
	{attribute addProperty Name "<#MANUAL#>"}
    {attribute addProperty ToolTip "<#Start manual/Service mode#>"}	
    _manualTask : CU00xManualTask(THIS^);
	{attribute addProperty Name "<#GROUND#>"}
	{attribute addProperty ToolTip "<#Brings the device into basic position.#>"}
	_groundTask : CU00xGroundTask(THIS^, TcoCore.eRestoreMode.None);
	{attribute addProperty Name "<#AUTOMAT#>"}
	{attribute addProperty ToolTip "<#Starts automatic sequence. Before start you need to perform grounding sequence.#>"}	
	_automatTask : CU00xAutomatTask(THIS^, TcoCore.eRestoreMode.None);     
	{attribute addProperty Name "<#SUSPEND PROCESS#>"}
    {attribute addProperty ToolTip "<#Starts suspend sequence of process(automatic,ground sequence).#>"}	
    _suspendTask : CU00xSuspendTask(THIS^, TcoCore.eRestoreMode.None);     
	{attribute addProperty Name "<#RECOVER PROCESS#>"}
    {attribute addProperty ToolTip "<#Starts suspend sequence of process(automatic,ground sequence).#>"}	
    _recoverTask : CU00xRecoverTask(THIS^, TcoCore.eRestoreMode.None);     
  	
	{attribute addProperty Name "<#Test positions#>"}
	_positions : Cu00xTestPositions(THIS^);

	{attribute addProperty Name "<#Test multi positions#>"}
	_positionsMulti : CU00xTestMultiPositions(THIS^);
END_VAR

THIS^.CuId := eStations.CU00x;



(*
	This controlled unit's component initialization.
*)

THIS^.InitializeComponents();

(*
	This controlled unit process data crud operations handler.
	Control exchange of process data between this controlled unit and the data repository.
*)

_processData();
_productionPlaner();


(*
	
	Cu's Modes
	
*)

Automat();
Ground();
Manual();


_suspendTask();
_recoverTask();







(*
	When no mode is active 'Idle' method should be called.
	'NoMode' method shouls contain code that renders this cu idle. 
*)

IF NOT (AutomatTask.Task.Busy 
		OR GroundTask.Task.Busy
		OR ManualTask.Task.Busy) 
THEN
	Idle();
END_IF



(*
	Updates this controlled unit's information for the UI.
*)


UpdateInfo();

_cuProcessDataDisplay := ProcessDataManager.Data.CU00x;
_cuTechnologicalDataDisplay := Technology.TechnologicalSettings.Data.CU00x;

_settings.WarningCycleTime:= _cuTechnologicalDataDisplay.WarningCycleTime;
_settings.ErrorCycleTime:= _cuTechnologicalDataDisplay.ErrorCycleTime;
_settings.AnyRecurringFailure:= _cuTechnologicalDataDisplay.AnyRecurringFailure;
_settings.SameRecurringFailure:= _cuTechnologicalDataDisplay.SameRecurringFailure;

(*~
	<docu>
		<summary>
			Controls `automatic` mode of `CU00x`.
		</summary>
	</docu>
~*)
METHOD Automat
VAR_INPUT
END_VAR
(*
	Enable condition to start `automatTask`.
	Modify according your needs.
	[! 
	THIS IS NOT SAFETY CONDITION. THE SAFETY OF PRESONNEL AND EQUIPMENT MUST BE ENSURED BY ADDITIONAL MEANS 
	TO COMPLY WITH REGULATIONS
	]
*)


//_automatTask.Task.Enabled := (_groundTask.GroundDone OR  _automatTask.Task.Busy) AND THIS^.Technology.AllowAutomat();

(*
	Invokes `groundTask` from technology object.
*)

//IF(Technology.AutomatAllTask.Execute()) THEN _automatTask.Task.Invoke(); END_IF;

//IF(Technology.ForceStepMode()) THEN
 //	_automatTask.ModeController.Mode := eSequencerMode.StepMode;
//END_IF 



(*
	or use default behavior from abstraction
*)
	SUPER^.Automat();

(*

	Executes sequence of automatic mode.

*)

_automatTask();
END_METHOD

PROPERTY AutomatTask : REFERENCE TO CUBaseAutomat
GET
AutomatTask REF= _automatTask;
END_GET
END_PROPERTY

PROPERTY Components : REFERENCE TO CU00xComponents
GET
Components REF= _components;
END_GET
END_PROPERTY

(*~
	<docu>
		<summary>
			Controls `ground` mode of `CU00x`.
		</summary>
	</docu>
~*)
METHOD Ground : BOOL
VAR_INPUT
END_VAR
(*
	Enable condition to start `groundTask`.
	Modify according your needs.
	[! 
	THIS IS NOT SAFETY CONDITION. THE SAFETY OF PRESONNEL AND EQUIPMENT MUST BE ENSURED BY ADDITIONAL MEANS 
	TO COMPLY WITH REGULATIONS
	]
*)

//_groundTask.Task.Enabled :=  THIS^.Technology.AllowGround();

(*
	Invokes `groundTask` from technology object.
*)

//IF(Technology.GroundAllTask.Execute()) THEN _groundTask.Task.Invoke(); END_IF;


//IF _groundTask.GroundDone AND _groundTask.Task.Execute() THEN _groundTask.Restore();_groundTask.Task.Invoke();END_IF;


(*
	or use default behavior from abstraction
*)
	SUPER^.Ground();




(*

	Executes sequence of groundTask.

*)

_groundTask();
END_METHOD

PROPERTY GroundTask : REFERENCE TO CUBaseGround
GET
GroundTask REF= _groundTask;
END_GET
END_PROPERTY

(*~
	<docu>
		<summary>
			Code to be called cylically when `CU00x` idle; no other mode is active.
		</summary>
	</docu>
~*)
METHOD Idle : BOOL
END_METHOD

METHOD InitializeComponents : BOOL

VAR_INST
	tempBoolHome: BOOL;
	tempBoolWork: BOOL;
	tempBoolP4Home: BOOL;
	tempBoolP4Work: BOOL;

END_VAR
VAR

	Output: INT;
END_VAR
_components.VerticalPiston(inoAtHomePos:= GVL_iXlinker.IN.Channel_1.Input
, inoAtWorkPos := GVL_iXlinker.IN.Channel_2.Input,
	inoToHomePos := GVL_iXlinker.OUT.Channel_1.Output, inoToWorkPos := GVL_iXlinker.OUT.Channel_2.Output);
	
_components.HorizontalPiston(inoAtHomePos:= GVL_iXlinker.IN.Channel_5.Input, inoAtWorkPos := GVL_iXlinker.IN.Channel_6.Input,
	inoToHomePos := GVL_iXlinker.OUT.Channel_3.Output, inoToWorkPos := GVL_iXlinker.OUT.Channel_4.Output);

_components.IN1(inoSignal:= GVL_iXlinker.B10_1);
_components.IN2(inoSignal:= GVL_iXlinker.IN.Channel_2.Input);
_components.IN3(inoSignal:= GVL_iXlinker.EC.EC.IA1.Channel_1.Input);

_components.OUT1(inoSignal:= GVL_iXlinker.B20_1);
_components.OUT2(inoSignal:= GVL_iXlinker.OUT.Channel_2.Output);
_components.OUT3(inoSignal:= GVL_iXlinker.EC.EC.QA1.Channel_1.Output);

(*
components.Group1.horizontalCylinder(inoAtHomePos:=GVL_iXlinker.EC1.EK1200.IA1_EL1809.Channel_1.Input, 
							   inoAtWorkPos:=GVL_iXlinker.EC1.EK1200.IA1_EL1809.Channel_2.Input, 
							   inoToHomePos:=GVL_iXlinker.EC1.EK1200.IA1_EL1809.Channel_3.Input, 
							   inoToWorkPos:=GVL_iXlinker.EC1.EK1200.IA1_EL1809.Channel_4.Input);
Components.SingleAxis.Config.InfoTime:=T#4S;
Components.SingleAxis.Config.ErrorTime:=T#10S;



Components.SingleAxis(inEnable := ,
    inEnablePositive := ,
    inEnableNegative := ,
    inCalibrationCam := ,
    refAxis := GVL_iXlinker.Axis1,
	inoPositions:= _positions);
	
	

//Components.PickAndPlace();
//Components.PickAndPlace.Service();
		
Components.MultiAxis(inEnableAxis1 := ,
    inEnablePositiveAxis1 := ,
    inEnableNegativeAxis1 := ,
    inCalibrationCamAxis1 := ,
    refAxis1 := GVL_iXlinker.Axis1,
	inoPositions:= _positionsMulti);
	
			
//Components.PickAndPlace.Components.Manipulator(inEnableAxis1 := ,
//    inEnablePositiveAxis1 := ,
//    inEnableNegativeAxis1 := ,
//    inCalibrationCamAxis1 := ,
//    refAxis1 := GVL_iXlinker.Axis1,
//	inoPositions:= _positionsMulti);
*)
END_METHOD

(*~
	<docu>
		<summary>
			Controls `manual` mode of `CU00x`.
		</summary>
	</docu>
~*)
METHOD Manual : BOOL
VAR_INPUT
END_VAR
(*
	Enable condition to start `automatTask`.
	Modify according your needs.
	[! 
	THIS IS NOT SAFETY CONDITION. THE SAFETY OF PRESONNEL AND EQUIPMENT MUST BE ENSURED BY ADDITIONAL MEANS 
	TO COMPLY WITH REGULATIONS
	]
*)

	//_manualTask.Task.Enabled := THIS^.Technology.AllowManual();

	
(*
	or use default behavior from abstraction
*)
	SUPER^.Manual();
	

(*

	Executes sequence of manualTask.

*)
_manualTask();
END_METHOD

PROPERTY ManualTask : REFERENCE TO TcoTaskedService
GET
ManualTask REF= _manualTask;
END_GET
END_PROPERTY

PROPERTY ProductionPlanerTask : REFERENCE TO ProductionPlaner
GET
ProductionPlanerTask REF= _productionPlaner;
END_GET
END_PROPERTY

PROPERTY RecoverTask : REFERENCE TO CUBaseRecover
GET
RecoverTask REF= _recoverTask;
END_GET
END_PROPERTY

PROPERTY StatusInfo : REFERENCE TO CUBaseStatusInfo
GET
StatusInfo ref= _statusInfo;
END_GET
END_PROPERTY

PROPERTY SuspendTask : REFERENCE TO CUBaseSuspend
GET
SuspendTask REF= _suspendTask;
END_GET
END_PROPERTY

PROPERTY Technology : REFERENCE TO Technology
GET
VAR
    _technology : POINTER TO Technology;
END_VAR
IF __QUERYPOINTER(Parent, _technology) THEN // Check if _Parent is Station001
    Technology REF= _technology^;              // If the check is successful dereference a pointer. simlar to THIS^ or SUPER^
END_IF
END_GET
END_PROPERTY

END_FUNCTION_BLOCK

// ---- Abstractions/CUBase/CUBase.TcPOU
{attribute addProperty ShortName ""}
FUNCTION_BLOCK ABSTRACT CUBase EXTENDS TcoCore.TcoObject IMPLEMENTS ICUBase

VAR
    _cuId        : eStations;
    _processData : ProcessDataManager(THIS^);
	_groupInspection : TcoInspectors.TcoInspectionGroup(THIS^);
	{attribute addProperty Name "<#STATUS INFO#>"}
    _statusInfo  : CUBaseStatusInfo := (Parent := THIS^);
	_operatorInfo : OperatorInfo := (Parent := THIS^);
	_settings  : CUBaseSettings := (Parent := THIS^);
	_toggle: TcoUtilities.TcoBlinker(THIS^);
	_recurringFails:CuBaseRecurringFailures:=(Parent:=THIS^);
	_productionPlaner:ProductionPlaner(THIS^);
	
END_VAR

(*~
	<docu>
		<summary>
			Controls `automatic` mode of `CU00x`.
		</summary>
	</docu>
~*)
METHOD  Automat
VAR_INPUT
END_VAR
(*
	Enable condition to start `automatTask`.
	Modify according your needs.
	[! 
	THIS IS NOT SAFETY CONDITION. THE SAFETY OF PRESONNEL AND EQUIPMENT MUST BE ENSURED BY ADDITIONAL MEANS 
	TO COMPLY WITH REGULATIONS
	]
*)


AutomatTask.Task.Enabled := (GroundTask.GroundDone OR  AutomatTask.Task.Busy) AND THIS^.Technology.AllowAutomat();

(*
	Invokes `groundTask` from technology object.
*)

IF(Technology.AutomatAllTask.Execute()) THEN AutomatTask.Task.Invoke(); END_IF;

IF(Technology.ForceStepMode()) THEN
 	AutomatTask.ModeController.Mode := eSequencerMode.StepMode;
END_IF
END_METHOD

PROPERTY ABSTRACT AutomatTask : REFERENCE TO CUBaseAutomat
GET
END_GET
END_PROPERTY

PROPERTY  CreateEntityTask : TcoCore.ITcoTaskStatus
GET
CreateEntityTask := _processData._createTask;
END_GET
END_PROPERTY

PROPERTY CuId : eStations
GET
CuId := _cuId;
END_GET
SET
_cuId := CuId;
END_SET
END_PROPERTY

PROPERTY  DeleteEntityTask : TcoCore.ITcoTaskStatus
GET
DeleteEntityTask := _processData._deleteTask;
END_GET
END_PROPERTY

METHOD EntityFlowCloseForOperations : TcoCore.ITcoTaskStatus
VAR_IN_OUT
	Header : CuHeader; 
END_VAR
THIS^.FlagCloseEntity(Header);
EntityFlowCloseForOperations := THIS^.ProcessDataManager.Update(ProcessDataManager.Data._EntityId);
END_METHOD

METHOD EntityFlowCreateNew : TcoCore.ITcoTaskStatus
VAR_INPUT
	EntityId : STRING(255);	
END_VAR
VAR_IN_OUT
	Header : CuHeader;
END_VAR
THIS^.FlagCreateNewEntity(EntityId, Header);
EntityFlowCreateNew := THIS^.ProcessDataManager.Create(EntityId);
END_METHOD

METHOD EntityFlowDiscard : TcoCore.ITcoTaskStatus
VAR_INPUT
	EntityId : STRING(255);	
END_VAR
VAR_IN_OUT	
	Header : CuHeader; 
END_VAR
THIS^.FlagThrowAwayEntity(Header);
EntityFlowDiscard := THIS^.ProcessDataManager.Update(EntityId);
END_METHOD

METHOD EntityFlowFinalize : TcoCore.ITcoTaskStatus
VAR_IN_OUT
	Header : CuHeader; 
END_VAR
THIS^.FlagFinishEntity(Header);
EntityFlowFinalize := THIS^.ProcessDataManager.Update(ProcessDataManager.Data._EntityId);
END_METHOD

METHOD EntityFlowOpenForOperations : TcoCore.ITcoTaskStatus
VAR_INPUT
	Identifier : STRING(255);	
END_VAR
VAR_IN_OUT
	Header : CuHeader;
END_VAR
EntityFlowOpenForOperations := THIS^.ProcessDataManager.Read(Identifier);
THIS^.FlagOpenEntity(Identifier, Header);
END_METHOD

PROPERTY  ExistEntityTask : TcoCore.ITcoTaskStatus
GET
ExistEntityTask := _processData._idExistsTask;
END_GET
END_PROPERTY

METHOD PRIVATE FlagCloseEntity : BOOL
VAR_IN_OUT
	Header : CuHeader; 
END_VAR
THIS^.ProcessDataManager.Data.EntityHeader.LastStation := THIS^.CuId;

IF(THIS^.ProcessDataManager.Data.EntityHeader.Results.Result = TcoInspectors.eOverallResult.Failed) THEN	
	THIS^.ProcessDataManager.Data.EntityHeader.NextStation := Header.NextOnFailed;
ELSIF(THIS^.ProcessDataManager.Data.EntityHeader.Results.Result = TcoInspectors.eOverallResult.Passed) THEN
	THIS^.ProcessDataManager.Data.EntityHeader.NextStation := Header.NextOnPassed;
ELSIF(THIS^.ProcessDataManager.Data.EntityHeader.Results.Result = TcoInspectors.eOverallResult.InProgress) THEN
	THIS^.ProcessDataManager.Data.EntityHeader.NextStation := Header.NextOnPassed;
END_IF

THIS^.ProcessDataManager.Data.EntityHeader.OpenOn := eStations.NONE;
Header.CycleTime := THIS^._statusInfo.CurrentCycleTime;
Header.CleanLoopTime := THIS^._statusInfo.CurrentCleanCycleTime;
Header.OperationsEnded := Context.RealTimeClock.NowLocal();
Header.Operator := _operatorInfo.UserName;
END_METHOD

METHOD PRIVATE FlagCreateNewEntity : BOOL
VAR_INPUT
	Identifier : STRING(255);	
END_VAR
VAR_IN_OUT
	Header : CuHeader;
END_VAR
THIS^.ProcessDataManager.Data.EntityHeader.Results.Result := TcoInspectors.eOverallResult.InProgress;
THIS^.ProcessDataManager.Data._EntityId := Identifier;
THIS^.ProcessDataManager.Data.EntityHeader.WasReset := FALSE;
END_METHOD

METHOD PRIVATE FlagFinishEntity : BOOL
VAR_IN_OUT
	Header : CuHeader; 
END_VAR
THIS^.ProcessDataManager.Data.EntityHeader.LastStation := THIS^.CuId;

IF(THIS^.ProcessDataManager.Data.EntityHeader.Results.Result = TcoInspectors.eOverallResult.InProgress) THEN
	THIS^.ProcessDataManager.Data.EntityHeader.Results.Result := TcoInspectors.eOverallResult.Passed;
END_IF

IF(THIS^.ProcessDataManager.Data.EntityHeader.Results.Result = TcoInspectors.eOverallResult.Failed) THEN	
	THIS^.ProcessDataManager.Data.EntityHeader.NextStation := Header.NextOnFailed;
ELSIF(THIS^.ProcessDataManager.Data.EntityHeader.Results.Result = TcoInspectors.eOverallResult.Passed) THEN
	THIS^.ProcessDataManager.Data.EntityHeader.NextStation := Header.NextOnPassed;
END_IF

THIS^.ProcessDataManager.Data.EntityHeader.OpenOn := eStations.NONE;

Header.CycleTime := THIS^._statusInfo.CurrentCycleTime;
Header.CleanLoopTime := THIS^._statusInfo.CurrentCleanCycleTime;
Header.OperationsEnded := Context.RealTimeClock.NowLocal();
Header.Operator := _operatorInfo.UserName;
END_METHOD

METHOD PRIVATE FlagOpenEntity : BOOL
VAR_INPUT
	Identifier : STRING(255);	
END_VAR
VAR_IN_OUT
	Header : CuHeader;
END_VAR
Header.Operator := _operatorInfo.UserName;
Header.OperationsStarted := Context.RealTimeClock.NowLocal();
THIS^.ProcessDataManager.Data.EntityHeader.Results.Result := TcoInspectors.eOverallResult.InProgress;
THIS^.ProcessDataManager.Data._EntityId := Identifier;
THIS^.ProcessDataManager.Data.EntityHeader.OpenOn := THIS^.CuId;
THIS^.ProcessDataManager.Data.EntityHeader.WasReset := FALSE;
END_METHOD

METHOD PRIVATE FlagThrowAwayEntity : BOOL
VAR_IN_OUT	
	CuHeader : CuHeader; 
END_VAR
IF(THIS^.ProcessDataManager.Data.EntityHeader.OpenOn <> eStations.NONE) THEN
	THIS^.ProcessDataManager.Data.EntityHeader.LastStation := THIS^.CuId;
	THIS^.ProcessDataManager.Data.EntityHeader.NextStation := CuHeader.NextOnFailed;
	THIS^.ProcessDataManager.Data.EntityHeader.Results.Result := TcoInspectors.eOverallResult.Failed;
	THIS^.ProcessDataManager.Data.EntityHeader.WasReset := TRUE;
END_IF;
END_METHOD

(*~
	<docu>
		<summary>
			Controls `ground` mode of `CU00x`.
		</summary>
	</docu>
~*)
METHOD Ground : BOOL
VAR_INPUT
END_VAR
(*
	Enable condition to start `groundTask`.
	Modify according your needs.
	[! 
	THIS IS NOT SAFETY CONDITION. THE SAFETY OF PRESONNEL AND EQUIPMENT MUST BE ENSURED BY ADDITIONAL MEANS 
	TO COMPLY WITH REGULATIONS
	]
*)

GroundTask.Task.Enabled :=  THIS^.Technology.AllowGround();

(*
	Invokes `groundTask` from technology object.
*)


IF(Technology.GroundAllTask.Execute()) THEN GroundTask.Restore();GroundTask.Task.Invoke(); END_IF;


IF GroundTask.GroundDone AND GroundTask.Task.Execute() THEN GroundTask.Restore();GroundTask.Task.Invoke();END_IF;
END_METHOD

PROPERTY ABSTRACT GroundTask : REFERENCE TO CUBaseGround
GET
END_GET
END_PROPERTY

PROPERTY FINAL GroupInspection : REFERENCE TO TcoInspectionGroup
GET
GroupInspection REF= _groupInspection;
END_GET
END_PROPERTY

(*~
	<docu>
		<summary>
			Code to be called cylically when `CU00x` idle; no other mode is active.
		</summary>
	</docu>
~*)
METHOD Idle : BOOL
END_METHOD

(*~
	<docu>
		<summary>
			Controls `manual` mode of `CU00x`.
		</summary>
	</docu>
~*)
METHOD Manual : BOOL
VAR_INPUT
END_VAR
(*
	Enable condition to start `automatTask`.
	Modify according your needs.
	[! 
	THIS IS NOT SAFETY CONDITION. THE SAFETY OF PRESONNEL AND EQUIPMENT MUST BE ENSURED BY ADDITIONAL MEANS 
	TO COMPLY WITH REGULATIONS
	]
*)

ManualTask.Task.Enabled := THIS^.Technology.AllowManual();
END_METHOD

PROPERTY ABSTRACT ManualTask : REFERENCE TO TcoTaskedService
GET
END_GET
END_PROPERTY

PROPERTY FINAL ProcessDataManager : REFERENCE TO ProcessDataManager
GET
ProcessDataManager REF= _processData;
END_GET
END_PROPERTY

PROPERTY  ReadEntityTask : TcoCore.ITcoTaskStatus
GET
ReadEntityTask := _processData._readTask;
END_GET
END_PROPERTY

PROPERTY ABSTRACT RecoverTask : REFERENCE TO CUBaseRecover
GET
END_GET
END_PROPERTY

PROPERTY RecurringFails : REFERENCE TO CuBaseRecurringFailures
GET
RecurringFails REF= _recurringFails;
END_GET
END_PROPERTY

PROPERTY ABSTRACT StatusInfo : REFERENCE TO CUBaseStatusInfo
GET
END_GET
END_PROPERTY

PROPERTY ABSTRACT SuspendTask : REFERENCE TO CUBaseSuspend
GET
END_GET
END_PROPERTY

PROPERTY Technology : REFERENCE TO Technology
GET
VAR
    _technology : POINTER TO Technology;
END_VAR
IF __QUERYPOINTER(Parent, _technology) THEN // Check if _Parent is Station001
    Technology REF= _technology^;              // If the check is successful dereference a pointer. simlar to THIS^ or SUPER^
END_IF
END_GET
END_PROPERTY

PROPERTY  UpdateEntityTask : TcoCore.ITcoTaskStatus
GET
UpdateEntityTask := _processData._updateTask;
END_GET
END_PROPERTY

METHOD UpdateInfo : BOOL
VAR_INPUT
END_VAR
_toggle(inOffTime:=T#500MS,inOnTime:=T#500MS);

_statusInfo.State := eCUState.None;

IF _statusInfo.CurrentCycleTime  >= _settings.WarningCycleTime
	AND _statusInfo.CurrentCycleTime  < _settings.ErrorCycleTime THEN
	_statusInfo.State:= eCUState.HasWarning;
ELSIF _statusInfo.CurrentCycleTime   >= _settings.ErrorCycleTime THEN
	_statusInfo.State := eCUState.HasError;
END_IF; 


IF _toggle.IsOff THEN
	_statusInfo.State := eCUState.None;
END_IF



IF AutomatTask.Task.Busy THEN
    _statusInfo.Mode                   := eCUMode.AutomatMode;
    _statusInfo.CurrentTaskDescription := '<#AUTOMAT#>';
    _statusInfo.CurrentCycleTime       := AutomatTask._SequenceElapsedTime;
	_statusInfo.CurrentCleanCycleTime  := T#0S;

	IF AutomatTask._startCleanCycleTime<>T#0S AND AutomatTask._stopCleanCycleTime=T#0S  THEN
		_statusInfo.CurrentCleanCycleTime  := AutomatTask._SequenceElapsedTime-AutomatTask._startCleanCycleTime;
	ELSIF AutomatTask._stopCleanCycleTime<>T#0S  THEN
		_statusInfo.CurrentCleanCycleTime  := AutomatTask._stopCleanCycleTime-AutomatTask._startCleanCycleTime;
	ELSE
		_statusInfo.CurrentCleanCycleTime :=AutomatTask._startCleanCycleTime;
	END_IF;
	
	_statusInfo.AverageCycleTime	   := AutomatTask.AverageCycleTime;
	_statusInfo.AverageCleanCycleTime  := AutomatTask.AverageCleanCycleTime;
    _statusInfo.CurrentUid             := AutomatTask.CurrentStep.ID;
    _statusInfo.CurrentOperation       := AutomatTask.CurrentStep.Description;
    _statusInfo.CurrentIsInStepMode    := AutomatTask._modeController._mode = eSequencerMode.StepMode;
ELSIF GroundTask.Task.Busy THEN
    _statusInfo.Mode := eCUMode.GroundMode;
	_statusInfo.CurrentTaskDescription := '<#GROUND#>';
    _statusInfo.CurrentCycleTime       := GroundTask._SequenceElapsedTime;
	_statusInfo.CurrentCleanCycleTime := T#0S;
	_statusInfo.AverageCycleTime	   := GroundTask.AverageCycleTime;
	_statusInfo.AverageCleanCycleTime  := T#0S;
    _statusInfo.CurrentUid             := GroundTask.CurrentStep.ID;
    _statusInfo.CurrentOperation       := GroundTask.CurrentStep.Description;
    _statusInfo.CurrentIsInStepMode    := GroundTask._modeController._mode = eSequencerMode.StepMode;
ELSIF THIS^.ManualTask.Busy THEN
    _statusInfo.Mode := eCUMode.ManualMode;
	_statusInfo.CurrentTaskDescription := '<#MANUAL#>';
	_statusInfo.State := eCUState.None;
	_statusInfo.CurrentIsInStepMode    := FALSE;

ELSIF THIS^.GroundTask.Task.Done THEN
	_statusInfo.CurrentTaskDescription := '<#READY TO START#>';
	_statusInfo.Mode := eCUMode.GroundModeDone;
	_statusInfo.CurrentCycleTime       := GroundTask._SequenceElapsedTime;
    _statusInfo.CurrentUid             := GroundTask.CurrentStep.ID;
    _statusInfo.CurrentOperation       := GroundTask.CurrentStep.Description;
    _statusInfo.CurrentIsInStepMode    := GroundTask._modeController._mode = eSequencerMode.StepMode;
	_statusInfo.State := eCUState.None;

ELSE
    _statusInfo.Mode := eCUMode.NoMode;	
	_statusInfo.CurrentTaskDescription := '<#IDLE#>';
	_statusInfo.CurrentCycleTime       := T#0S;
    _statusInfo.CurrentUid             := 0;
    _statusInfo.CurrentOperation       := '';
    _statusInfo.CurrentIsInStepMode    := FALSE;
	_statusInfo.State := eCUState.None;
END_IF
END_METHOD

END_FUNCTION_BLOCK

// ---- Abstractions/CUBase/RemoteTasks/ProductionPlaner.TcPOU
FUNCTION_BLOCK PUBLIC ProductionPlaner EXTENDS TcoCore.TcoRemoteTask
VAR_INPUT
END_VAR
VAR_OUTPUT
END_VAR
VAR
	_productonPlanCompleted: BOOL;
	_productionPlanIsEmpty: BOOL;
	_requiredProcessSettings: STRING;
END_VAR

super^();

PROPERTY PUBLIC ProductionPlanCompleted : bool
GET
ProductionPlanCompleted:=_productonPlanCompleted;
END_GET
END_PROPERTY

PROPERTY PUBLIC ProductionPlanIsEmpty : bool
GET
ProductionPlanIsEmpty:=_productionPlanIsEmpty;
END_GET
END_PROPERTY

PROPERTY RequiredProcessSettingsId : string
GET
RequiredProcessSettingsId:=_requiredProcessSettings;
END_GET
END_PROPERTY

(*~
	<docu>
		<summary>
			Restores this instance to the Ready state. Can be called explicitly or from within one of the restore mechanisms.
			<para>
				See also <see cref="PlcDocu.TcoCore.TcoTask.AutoRestorable()"/>
			</para>
		</summary>			
	</docu>	
~*)
METHOD Restore : ITcoRestorable
SUPER^.Restore();
_productonPlanCompleted:=FALSE;
_productionPlanIsEmpty:=FALSE;
_requiredProcessSettings:='';
END_METHOD

END_FUNCTION_BLOCK

// ---- Abstractions/CUBase/Tasks/CUBaseAutomat.TcPOU
FUNCTION_BLOCK ABSTRACT CUBaseAutomat EXTENDS TcoTaskedSequencer
VAR
    _dialog : TcoCore.TcoDialog(THIS^);
    _dialogCustomized : TcoCore.TcoCustomizedDialog(THIS^);
    _dialogWithInput : TcoCore.TcoInputDialog(THIS^);
END_VAR

(*~
	<docu>
		<summary>
			Stores the data from this controlled unit into the repository. In addition modifies entity header and controlled unit header.									
		</summary>
	</docu>
~*)
METHOD DataEntityClose
VAR_INPUT
	(*~
	<docu>
		<summary>
			The unique step id definition.
		</summary>			
	</docu>	
	~*)
	inStepID : INT;
	(*~
	<docu>
		<summary>
			If input enum is set to InvokeAndWaitDone  operation will  wait until task reaches the ```Done``` state .
			If input enum is set to InvokeOnly results return True when  task reaches the ```Busy``` state . Later is recomended (neccessary) to check  task  ```Done``` state  , check  task  status.
		</summary>			
	</docu>	
	~*)
	InvokeAction: eDataEntityInvokeType;
END_VAR
VAR_IN_OUT
	Header : CuHeader; 
END_VAR
IF (Step(inStepID,TRUE, 'CLOSE ENTITY DATA')) THEN
    //-------------------------------------		
	CASE InvokeAction OF
		eDataEntityInvokeType.InvokeAndWaitDone: 
				StepCompleteWhen(THIS^.StationBase.EntityFlowCloseForOperations(Header).Done);
		eDataEntityInvokeType.InvokeOnly: 
				StepCompleteWhen(THIS^.StationBase.EntityFlowCloseForOperations(Header).Busy);	
	END_CASE;			   		    				
    //-------------------------------------
END_IF
END_METHOD

(*~
	<docu>
		<summary>
			Creates new record in the repository with given EntityId and populates with the current controlled units data.
			In addition modifies entity header and controlled unit header.									
		</summary>
	</docu>
~*)
METHOD DataEntityCreateNew
VAR_INPUT	
	inStepID : INT;
	EntityId : STRING(255);
END_VAR

VAR_IN_OUT
	Header: CuHeader;
END_VAR
IF (Step(inStepID, TRUE, 'CREATE NEW ENTITY DATA')) THEN
    //-------------------------------------		
	StepCompleteWhen(THIS^.StationBase.EntityFlowCreateNew(EntityId, Header).Done);				   		    				
    //-------------------------------------
END_IF
END_METHOD

METHOD DataEntityDiscard
VAR_INPUT	
	inStepID : INT;
	EntityId : STRING(255);
END_VAR
VAR_IN_OUT
	Header: CuHeader;
END_VAR
IF (Step(inStepID, TRUE, 'DISCARD ENTITY DATA')) THEN
    //-------------------------------------		
	StepCompleteWhen(THIS^.StationBase.EntityFlowDiscard(EntityId, Header).Done);				   		    				
    //-------------------------------------
END_IF
END_METHOD

(*~
	<docu>
		<summary>
			Stores data of this controlled unit into the repository.
			In addition modifies entity header and controlled unit header.
			Finalize will set the comprehensive result from InProgress to Passed. 
			If the comprehensive result is Failed the finalizing will not modify the result.									
		</summary>
	</docu>
~*)
METHOD DataEntityFinalize : BOOL
VAR_INPUT
	(*~
	<docu>
		<summary>
			The unique step id definition.
		</summary>			
	</docu>	
	~*)
	inStepID : INT;
	(*~
	<docu>
		<summary>
			If input enum is set to InvokeAndWaitDone  operation will  wait until task reaches the ```Done``` state .
			If input enum is set to InvokeOnly results return True when  task reaches the ```Busy``` state . This option is used when we need to reduce cycle time. Later is recomended (neccessary) to check  task  ```Done``` state  , check  task  status.
		</summary>			
	</docu>	
	~*)
	InvokeAction: eDataEntityInvokeType;
END_VAR
VAR_IN_OUT
	Header: CuHeader;
END_VAR
IF (Step(inStepID,TRUE, 'FINALIZE ENTITY DATA')) THEN
    //-------------------------------------		
		CASE InvokeAction OF
		eDataEntityInvokeType.InvokeAndWaitDone: 
				StepCompleteWhen(THIS^.StationBase.EntityFlowFinalize(Header).Done);
		eDataEntityInvokeType.InvokeOnly: 
				StepCompleteWhen(THIS^.StationBase.EntityFlowFinalize(Header).Busy);	
	END_CASE;			   		    				
	StepCompleteWhen(THIS^.StationBase.EntityFlowFinalize(Header).Done );				   		    				
    //-------------------------------------
END_IF
END_METHOD

(*~
	<docu>
		<summary>
			Retrieves the data with given EntityId from the repository. In addition modifies entity header and controlled unit header.									
		</summary>
	</docu>
~*)
METHOD DataEntityOpen
VAR_INPUT
	(*~
	<docu>
		<summary>
			The unique step id definition.
		</summary>			
	</docu>	
	~*)
	inStepID : INT;
	(*~
	<docu>
		<summary>
			The definition of jump sptep.Usage of this jump step is when entity does not belong to the Controled unit.
		</summary>			
	</docu>	
	~*)
	inReqStepId: INT;
	inEntityId : STRING(255);
END_VAR
VAR_IN_OUT
	CuHeader: CuHeader;
END_VAR
IF (Step(inStepID, TRUE, 'OPEN ENTITY DATA')) THEN
    //-------------------------------------		
    IF THIS^.StationBase.EntityFlowOpenForOperations(inEntityId, CuHeader).Done THEN
        IF THIS^.StationBase.ProcessDataManager.Data.EntityHeader.IsEmpty THEN
            RequestStep(inReqStepId);
        ELSIF EntityDoesBelong() THEN
            CompleteStep();
        ELSE
            RequestStep(inReqStepId);
        END_IF
    END_IF;
    //-------------------------------------
END_IF
END_METHOD

METHOD EntityDoesBelong : BOOL
VAR_INPUT
END_VAR
EntityDoesBelong:=THIS^.StationBase.ProcessDataManager.Data.EntityHeader.NextStation = THIS^.StationBase.CuId;
END_METHOD

METHOD PUBLIC  HideAllDialogs
VAR_INPUT
END_VAR
_dialog.Restore();
_dialogWithInput.Restore();
_dialogCustomized.Restore();
END_METHOD

METHOD MonitorAnyRecurringFailure
VAR_INPUT
	(*~
	<docu>
		<summary>
			The unique step id definition.
		</summary>			
	</docu>	
	~*)
	inStepID : INT;
	(*~
	<docu>
		<summary>
			The step enable condition.
		</summary>			
	</docu>	
	~*)
	inEnableStep :BOOL;
	inResult : TcoComprehensiveResult;
END_VAR
IF (Step(inStepID,inEnableStep, 'MONITOR ANY RECURRING FAILURE IN SEQUENCE')) THEN
    //-------------------------------------		
	
